LIN {X -0.127,Y -423.917,Z 1358.586,A 0.000,B 0.000,C 90.000,E1 105.536} C_DIS
LIN {X 0.148,Y -443.072,Z 1358.574,A 0.000,B 0.000,C 90.000,E1 103.355} C_DIS
LIN {X 0.036,Y -463.165,Z 1358.563,A 0.000,B 0.000,C 90.000,E1 101.366} C_DIS
LIN {X 0.203,Y -481.163,Z 1358.554,A 0.000,B 0.000,C 90.000,E1 99.726} C_DIS
LIN {X 0.205,Y -483.225,Z 1358.553,A 0.000,B 0.000,C 90.000,E1 99.500} C_DIS
LIN {X -0.191,Y -484.795,Z 1358.552,A 0.000,B 0.000,C 90.000,E1 99.321} C_DIS
LIN {X 0.175,Y -486.110,Z 1358.550,A 0.000,B 0.000,C 90.000,E1 99.029} C_DIS
LIN {X -0.014,Y -487.078,Z 1358.549,A 0.000,B 0.000,C 90.000,E1 98.803} C_DIS
LIN {X 0.255,Y -488.153,Z 1358.546,A 0.000,B 0.000,C 90.000,E1 98.276} C_DIS
LIN {X -0.026,Y -488.220,Z 1358.543,A 0.000,B 0.000,C 90.000,E1 97.814} C_DIS
LIN {X 0.184,Y -487.293,Z 1358.541,A 0.000,B 0.000,C 90.000,E1 97.296} C_DIS
LIN {X -0.088,Y -485.213,Z 1358.538,A 0.000,B 0.000,C 90.000,E1 96.834} C_DIS
LIN {X 0.116,Y -481.753,Z 1358.535,A 0.000,B 0.000,C 90.000,E1 96.315} C_DIS
LIN {X 0.079,Y -471.298,Z 1358.527,A 0.000,B 0.000,C 90.000,E1 94.821} C_DIS
LIN {X -0.125,Y -461.369,Z 1358.518,A 0.000,B 0.000,C 90.000,E1 93.326} C_DIS
LIN {X -0.174,Y -441.725,Z 1358.501,A 0.000,B 0.000,C 90.000,E1 90.229} C_DIS
LIN {X 0.004,Y -428.339,Z 1358.488,A 0.000,B 0.000,C 90.000,E1 87.822} C_DIS
LIN {X 0.068,Y -418.056,Z 1358.477,A 0.000,B 0.000,C 90.000,E1 85.927} C_DIS
LIN {X -0.091,Y -407.688,Z 1358.467,A 0.000,B 0.000,C 90.000,E1 84.033} C_DIS
LIN {X -0.013,Y -398.629,Z 1358.458,A 0.000,B 0.000,C 90.000,E1 82.356} C_DIS
LIN {X -0.094,Y -389.359,Z 1358.448,A 0.000,B 0.000,C 90.000,E1 80.679} C_DIS
LIN {X 0.168,Y -379.910,Z 1358.439,A 0.000,B 0.000,C 90.000,E1 78.926} C_DIS
LIN {X -0.108,Y -370.271,Z 1358.429,A 0.000,B 0.000,C 90.000,E1 77.229} C_DIS
LIN {X -0.144,Y -358.777,Z 1358.417,A 0.000,B 0.000,C 90.000,E1 75.172} C_DIS
LIN {X 0.162,Y -348.864,Z 1358.407,A 0.000,B 0.000,C 90.000,E1 73.323} C_DIS
LIN {X -0.054,Y -337.184,Z 1358.396,A 0.000,B 0.000,C 90.000,E1 71.221} C_DIS
LIN {X -0.015,Y -323.949,Z 1358.382,A 0.000,B 0.000,C 90.000,E1 68.720} C_DIS
LIN {X -0.098,Y -308.256,Z 1358.364,A 0.000,B 0.000,C 90.000,E1 65.537} C_DIS
LIN {X -0.142,Y -298.262,Z 1358.351,A 0.000,B 0.000,C 90.000,E1 63.256} C_DIS
LIN {X 0.106,Y -288.081,Z 1358.336,A 0.000,B 0.000,C 90.000,E1 60.539} C_DIS
LIN {X -0.039,Y -281.281,Z 1358.325,A 0.000,B 0.000,C 90.000,E1 58.535} C_DIS
LIN {X -0.059,Y -271.116,Z 1358.306,A 0.000,B 0.000,C 90.000,E1 55.102} C_DIS
LIN {X 0.096,Y -263.450,Z 1358.291,A 0.000,B 0.000,C 90.000,E1 52.271} C_DIS
LIN {X 0.038,Y -254.301,Z 1358.271,A 0.000,B 0.000,C 90.000,E1 48.728} C_DIS
LIN {X 0.156,Y -247.369,Z 1358.255,A 0.000,B 0.000,C 90.000,E1 45.810} C_DIS
LIN {X 0.070,Y -239.383,Z 1358.234,A 0.000,B 0.000,C 90.000,E1 42.162} C_DIS
LIN {X -0.044,Y -232.253,Z 1358.214,A 0.000,B 0.000,C 90.000,E1 38.463} C_DIS
LIN {X -0.076,Y -225.922,Z 1358.193,A 0.000,B 0.000,C 90.000,E1 34.692} C_DIS
LIN {X -0.007,Y -220.570,Z 1358.171,A 0.000,B 0.000,C 90.000,E1 30.846} C_DIS
LIN {X -0.100,Y -216.212,Z 1358.150,A 0.000,B 0.000,C 90.000,E1 27.001} C_DIS
LIN {X 0.020,Y -212.299,Z 1358.124,A 0.000,B 0.000,C 90.000,E1 22.280} C_DIS
LIN {X -0.044,Y -209.772,Z 1358.102,A 0.000,B 0.000,C 90.000,E1 18.362} C_DIS
LIN {X -0.011,Y -207.919,Z 1358.084,A 0.000,B 0.000,C 90.000,E1 15.190} C_DIS
LIN {X 0.102,Y -205.787,Z 1358.062,A 0.000,B 0.000,C 90.000,E1 11.186} C_DIS
LIN {X -0.089,Y -204.193,Z 1358.045,A 0.000,B 0.000,C 90.000,E1 8.049} C_DIS
LIN {X 0.006,Y -202.797,Z 1358.027,A 0.000,B 0.000,C 90.000,E1 4.821} C_DIS
LIN {X -0.036,Y -200.987,Z 1357.997,A 0.000,B 0.000,C 90.000,E1 359.542} C_DIS
LIN {X -0.090,Y -200.235,Z 1357.966,A 0.000,B 0.000,C 90.000,E1 353.913} C_DIS
LIN {X -0.015,Y -201.594,Z 1357.921,A 0.000,B 0.000,C 90.000,E1 345.825} C_DIS
LIN {X 0.033,Y -204.564,Z 1357.890,A 0.000,B 0.000,C 90.000,E1 340.188} C_DIS
LIN {X 0.003,Y -208.549,Z 1357.863,A 0.000,B 0.000,C 90.000,E1 335.409} C_DIS
LIN {X 0.071,Y -213.049,Z 1357.841,A 0.000,B 0.000,C 90.000,E1 331.435} C_DIS
LIN {X 0.022,Y -218.800,Z 1357.820,A 0.000,B 0.000,C 90.000,E1 327.533} C_DIS
LIN {X -0.119,Y -225.621,Z 1357.798,A 0.000,B 0.000,C 90.000,E1 323.703} C_DIS
LIN {X -0.088,Y -232.011,Z 1357.781,A 0.000,B 0.000,C 90.000,E1 320.642} C_DIS
LIN {X -0.106,Y -239.229,Z 1357.765,A 0.000,B 0.000,C 90.000,E1 317.634} C_DIS
LIN {X 0.024,Y -248.202,Z 1357.746,A 0.000,B 0.000,C 90.000,E1 314.271} C_DIS
LIN {X -0.125,Y -256.103,Z 1357.732,A 0.000,B 0.000,C 90.000,E1 311.757} C_DIS
LIN {X -0.027,Y -266.363,Z 1357.716,A 0.000,B 0.000,C 90.000,E1 308.874} C_DIS
LIN {X -0.018,Y -279.522,Z 1357.698,A 0.000,B 0.000,C 90.000,E1 305.724} C_DIS
LIN {X 0.063,Y -287.690,Z 1357.689,A 0.000,B 0.000,C 90.000,E1 303.992} C_DIS
LIN {X -0.121,Y -296.776,Z 1357.680,A 0.000,B 0.000,C 90.000,E1 302.339} C_DIS
LIN {X -0.078,Y -306.973,Z 1357.670,A 0.000,B 0.000,C 90.000,E1 300.669} C_DIS
LIN {X 0.082,Y -316.117,Z 1357.663,A 0.000,B 0.000,C 90.000,E1 299.333} C_DIS
LIN {X 0.050,Y -336.742,Z 1357.649,A 0.000,B 0.000,C 90.000,E1 296.796} C_DIS
LIN {X -0.056,Y -352.620,Z 1357.639,A 0.000,B 0.000,C 90.000,E1 295.027} C_DIS
LIN {X 0.023,Y -365.723,Z 1357.631,A 0.000,B 0.000,C 90.000,E1 293.567} C_DIS
LIN {X 0.066,Y -375.959,Z 1357.625,A 0.000,B 0.000,C 90.000,E1 292.408} C_DIS
LIN {X -0.001,Y -388.536,Z 1357.616,A 0.000,B 0.000,C 90.000,E1 290.972} C_DIS
LIN {X -0.014,Y -403.296,Z 1357.607,A 0.000,B 0.000,C 90.000,E1 289.268} C_DIS
LIN {X 0.119,Y -417.975,Z 1357.598,A 0.000,B 0.000,C 90.000,E1 287.583} C_DIS
LIN {X 0.090,Y -427.465,Z 1357.592,A 0.000,B 0.000,C 90.000,E1 286.496} C_DIS
LIN {X -0.127,Y -434.044,Z 1357.587,A 0.000,B 0.000,C 90.000,E1 285.717} C_DIS
LIN {X 0.011,Y -440.022,Z 1357.583,A 0.000,B 0.000,C 90.000,E1 284.898} C_DIS
LIN {X -0.102,Y -445.273,Z 1357.578,A 0.000,B 0.000,C 90.000,E1 284.120} C_DIS
LIN {X 0.150,Y -449.712,Z 1357.574,A 0.000,B 0.000,C 90.000,E1 283.300} C_DIS
LIN {X 0.014,Y -453.341,Z 1357.570,A 0.000,B 0.000,C 90.000,E1 282.535} C_DIS
LIN {X -0.097,Y -456.212,Z 1357.565,A 0.000,B 0.000,C 90.000,E1 281.771} C_DIS
LIN {X -0.012,Y -457.679,Z 1357.563,A 0.000,B 0.000,C 90.000,E1 281.243} C_DIS
LIN {X 0.082,Y -458.764,Z 1357.560,A 0.000,B 0.000,C 90.000,E1 280.715} C_DIS
LIN {X 0.100,Y -459.438,Z 1357.557,A 0.000,B 0.000,C 90.000,E1 280.197} C_DIS
LIN {X 0.207,Y -459.649,Z 1357.554,A 0.000,B 0.000,C 90.000,E1 279.670} C_DIS
LIN {X -0.212,Y -459.367,Z 1357.551,A 0.000,B 0.000,C 90.000,E1 279.208} C_DIS
LIN {X -0.104,Y -458.592,Z 1357.548,A 0.000,B 0.000,C 90.000,E1 278.681} C_DIS
LIN {X -0.068,Y -457.352,Z 1357.545,A 0.000,B 0.000,C 90.000,E1 278.163} C_DIS
LIN {X -0.035,Y -455.526,Z 1357.542,A 0.000,B 0.000,C 90.000,E1 277.644} C_DIS
LIN {X -0.006,Y -453.175,Z 1357.540,A 0.000,B 0.000,C 90.000,E1 277.125} C_DIS
LIN {X 0.005,Y -450.289,Z 1357.537,A 0.000,B 0.000,C 90.000,E1 276.606} C_DIS
LIN {X 0.002,Y -446.827,Z 1357.534,A 0.000,B 0.000,C 90.000,E1 276.087} C_DIS
LIN {X -0.019,Y -442.576,Z 1357.531,A 0.000,B 0.000,C 90.000,E1 275.568} C_DIS
LIN {X -0.063,Y -437.339,Z 1357.528,A 0.000,B 0.000,C 90.000,E1 275.049} C_DIS
LIN {X 0.120,Y -431.246,Z 1357.525,A 0.000,B 0.000,C 90.000,E1 274.531} C_DIS
LIN {X -0.098,Y -424.898,Z 1357.523,A 0.000,B 0.000,C 90.000,E1 274.131} C_DIS
LIN {X 0.152,Y -418.457,Z 1357.521,A 0.000,B 0.000,C 90.000,E1 273.726} C_DIS
LIN {X -0.130,Y -412.038,Z 1357.519,A 0.000,B 0.000,C 90.000,E1 273.440} C_DIS
LIN {X 0.208,Y -405.345,Z 1357.517,A 0.000,B 0.000,C 90.000,E1 273.094} C_DIS
LIN {X -0.065,Y -395.236,Z 1357.515,A 0.000,B 0.000,C 90.000,E1 272.751} C_DIS
LIN {X 0.029,Y -388.350,Z 1357.514,A 0.000,B 0.000,C 90.000,E1 272.522} C_DIS
LIN {X -0.051,Y -381.280,Z 1357.513,A 0.000,B 0.000,C 90.000,E1 272.350} C_DIS
LIN {X 0.050,Y -373.704,Z 1357.512,A 0.000,B 0.000,C 90.000,E1 272.178} C_DIS
LIN {X -0.014,Y -364.873,Z 1357.511,A 0.000,B 0.000,C 90.000,E1 272.064} C_DIS
LIN {X -0.163,Y -352.105,Z 1357.511,A 0.000,B 0.000,C 90.000,E1 271.949} C_DIS
LIN {X 0.082,Y -339.041,Z 1357.510,A 0.000,B 0.000,C 90.000,E1 271.835} C_DIS
LIN {X 0.019,Y -330.015,Z 1357.510,A 0.000,B 0.000,C 90.000,E1 271.835} C_DIS
LIN {X -0.009,Y -181.290,Z 1357.510,A 0.000,B 0.000,C 90.000,E1 271.835} C_DIS
LIN {X 0.038,Y -181.580,Z 1357.502,A 0.000,B 0.000,C 90.000,E1 270.286} C_DIS
LIN {X -0.002,Y -180.908,Z 1357.475,A 0.000,B 0.000,C 90.000,E1 265.584} C_DIS
LIN {X 0.055,Y -180.783,Z 1357.471,A 0.000,B 0.000,C 90.000,E1 264.723} C_DIS
LIN {X -0.050,Y -178.880,Z 1357.443,A 0.000,B 0.000,C 90.000,E1 259.690} C_DIS
LIN {X 0.026,Y -175.923,Z 1357.414,A 0.000,B 0.000,C 90.000,E1 254.574} C_DIS
LIN {X -0.084,Y -174.622,Z 1357.405,A 0.000,B 0.000,C 90.000,E1 252.906} C_DIS
LIN {X 0.008,Y -171.603,Z 1357.381,A 0.000,B 0.000,C 90.000,E1 248.592} C_DIS
LIN {X -0.004,Y -167.825,Z 1357.357,A 0.000,B 0.000,C 90.000,E1 244.280} C_DIS
LIN {X 0.014,Y -166.549,Z 1357.347,A 0.000,B 0.000,C 90.000,E1 242.538} C_DIS
LIN {X -0.076,Y -162.546,Z 1357.323,A 0.000,B 0.000,C 90.000,E1 238.201} C_DIS
LIN {X -0.016,Y -161.223,Z 1357.313,A 0.000,B 0.000,C 90.000,E1 236.421} C_DIS
LIN {X 0.020,Y -157.229,Z 1357.289,A 0.000,B 0.000,C 90.000,E1 231.984} C_DIS
LIN {X 0.043,Y -155.955,Z 1357.279,A 0.000,B 0.000,C 90.000,E1 230.194} C_DIS
LIN {X 0.001,Y -152.207,Z 1357.254,A 0.000,B 0.000,C 90.000,E1 225.729} C_DIS
LIN {X 0.022,Y -150.452,Z 1357.239,A 0.000,B 0.000,C 90.000,E1 223.014} C_DIS
LIN {X 0.048,Y -147.178,Z 1357.214,A 0.000,B 0.000,C 90.000,E1 218.463} C_DIS
LIN {X 0.015,Y -145.196,Z 1357.193,A 0.000,B 0.000,C 90.000,E1 214.818} C_DIS
LIN {X 0.050,Y -142.335,Z 1357.163,A 0.000,B 0.000,C 90.000,E1 209.283} C_DIS
LIN {X -0.021,Y -141.723,Z 1357.152,A 0.000,B 0.000,C 90.000,E1 207.462} C_DIS
LIN {X -0.039,Y -139.479,Z 1357.116,A 0.000,B 0.000,C 90.000,E1 200.972} C_DIS
LIN {X -0.049,Y -138.976,Z 1357.101,A 0.000,B 0.000,C 90.000,E1 198.181} C_DIS
LIN {X 0.072,Y -138.331,Z 1357.054,A 0.000,B 0.000,C 90.000,E1 189.726} C_DIS
LIN {X -0.064,Y -139.432,Z 1357.007,A 0.000,B 0.000,C 90.000,E1 181.375} C_DIS
LIN {X 0.015,Y -140.958,Z 1356.976,A 0.000,B 0.000,C 90.000,E1 175.755} C_DIS
LIN {X -0.034,Y -142.713,Z 1356.956,A 0.000,B 0.000,C 90.000,E1 172.064} C_DIS
LIN {X 0.065,Y -145.090,Z 1356.930,A 0.000,B 0.000,C 90.000,E1 167.409} C_DIS
LIN {X 0.061,Y -147.715,Z 1356.910,A 0.000,B 0.000,C 90.000,E1 163.740} C_DIS
LIN {X 0.002,Y -150.372,Z 1356.890,A 0.000,B 0.000,C 90.000,E1 160.115} C_DIS
LIN {X 0.020,Y -153.800,Z 1356.869,A 0.000,B 0.000,C 90.000,E1 156.485} C_DIS
LIN {X 0.080,Y -157.211,Z 1356.849,A 0.000,B 0.000,C 90.000,E1 152.871} C_DIS
LIN {X 0.021,Y -161.376,Z 1356.830,A 0.000,B 0.000,C 90.000,E1 149.331} C_DIS
LIN {X 0.032,Y -165.578,Z 1356.810,A 0.000,B 0.000,C 90.000,E1 145.801} C_DIS
LIN {X 0.018,Y -170.499,Z 1356.791,A 0.000,B 0.000,C 90.000,E1 142.316} C_DIS
LIN {X 0.064,Y -175.379,Z 1356.771,A 0.000,B 0.000,C 90.000,E1 138.852} C_DIS
LIN {X -0.074,Y -181.003,Z 1356.753,A 0.000,B 0.000,C 90.000,E1 135.486} C_DIS
LIN {X 0.051,Y -186.431,Z 1356.734,A 0.000,B 0.000,C 90.000,E1 132.081} C_DIS
LIN {X 0.119,Y -191.058,Z 1356.720,A 0.000,B 0.000,C 90.000,E1 129.564} C_DIS
LIN {X 0.042,Y -196.843,Z 1356.702,A 0.000,B 0.000,C 90.000,E1 126.297} C_DIS
LIN {X 0.051,Y -199.194,Z 1356.695,A 0.000,B 0.000,C 90.000,E1 125.105} C_DIS
LIN {X 0.046,Y -308.858,Z 1356.695,A 0.000,B 0.000,C 90.000,E1 125.105} C_DIS
LIN {X -0.191,Y -311.436,Z 1356.695,A 0.000,B 0.000,C 90.000,E1 125.105} C_DIS
LIN {X -0.128,Y -315.472,Z 1356.694,A 0.000,B 0.000,C 90.000,E1 124.898} C_DIS
LIN {X -0.063,Y -317.840,Z 1356.693,A 0.000,B 0.000,C 90.000,E1 124.692} C_DIS
LIN {X 0.014,Y -321.665,Z 1356.690,A 0.000,B 0.000,C 90.000,E1 124.199} C_DIS
LIN {X 0.089,Y -323.434,Z 1356.688,A 0.000,B 0.000,C 90.000,E1 123.865} C_DIS
LIN {X -0.106,Y -324.810,Z 1356.686,A 0.000,B 0.000,C 90.000,E1 123.579} C_DIS
LIN {X -0.011,Y -336.372,Z 1356.669,A 0.000,B 0.000,C 90.000,E1 120.413} C_DIS
LIN {X -0.054,Y -348.165,Z 1356.654,A 0.000,B 0.000,C 90.000,E1 117.641} C_DIS
LIN {X 0.058,Y -361.406,Z 1356.638,A 0.000,B 0.000,C 90.000,E1 114.899} C_DIS
LIN {X 0.156,Y -374.481,Z 1356.625,A 0.000,B 0.000,C 90.000,E1 112.514} C_DIS
LIN {X -0.202,Y -388.879,Z 1356.612,A 0.000,B 0.000,C 90.000,E1 110.248} C_DIS
LIN {X 0.033,Y -404.701,Z 1356.600,A 0.000,B 0.000,C 90.000,E1 107.946} C_DIS
LIN {X 0.154,Y -422.057,Z 1356.587,A 0.000,B 0.000,C 90.000,E1 105.717} C_DIS
LIN {X -0.058,Y -441.070,Z 1356.575,A 0.000,B 0.000,C 90.000,E1 103.592} C_DIS
LIN {X 0.228,Y -461.105,Z 1356.564,A 0.000,B 0.000,C 90.000,E1 101.535} C_DIS
LIN {X -0.165,Y -481.566,Z 1356.554,A 0.000,B 0.000,C 90.000,E1 99.726} C_DIS
LIN {X -0.201,Y -483.525,Z 1356.553,A 0.000,B 0.000,C 90.000,E1 99.500} C_DIS
LIN {X -0.156,Y -485.019,Z 1356.551,A 0.000,B 0.000,C 90.000,E1 99.265} C_DIS
LIN {X 0.212,Y -486.241,Z 1356.550,A 0.000,B 0.000,C 90.000,E1 98.973} C_DIS
LIN {X 0.025,Y -487.133,Z 1356.549,A 0.000,B 0.000,C 90.000,E1 98.746} C_DIS
LIN {X -0.187,Y -488.080,Z 1356.546,A 0.000,B 0.000,C 90.000,E1 98.276} C_DIS
LIN {X 0.015,Y -488.028,Z 1356.543,A 0.000,B 0.000,C 90.000,E1 97.757} C_DIS
LIN {X 0.225,Y -486.975,Z 1356.540,A 0.000,B 0.000,C 90.000,E1 97.239} C_DIS
LIN {X 0.119,Y -486.024,Z 1356.539,A 0.000,B 0.000,C 90.000,E1 97.004} C_DIS
LIN {X -0.047,Y -484.730,Z 1356.538,A 0.000,B 0.000,C 90.000,E1 96.777} C_DIS
LIN {X 0.143,Y -470.717,Z 1356.526,A 0.000,B 0.000,C 90.000,E1 94.759} C_DIS
LIN {X -0.109,Y -460.779,Z 1356.518,A 0.000,B 0.000,C 90.000,E1 93.269} C_DIS
LIN {X 0.073,Y -442.697,Z 1356.502,A 0.000,B 0.000,C 90.000,E1 90.401} C_DIS
LIN {X -0.155,Y -429.271,Z 1356.489,A 0.000,B 0.000,C 90.000,E1 88.051} C_DIS
LIN {X -0.098,Y -419.002,Z 1356.479,A 0.000,B 0.000,C 90.000,E1 86.159} C_DIS
LIN {X -0.196,Y -408.662,Z 1356.468,A 0.000,B 0.000,C 90.000,E1 84.261} C_DIS
LIN {X -0.146,Y -399.649,Z 1356.459,A 0.000,B 0.000,C 90.000,E1 82.591} C_DIS
LIN {X -0.149,Y -390.407,Z 1356.449,A 0.000,B 0.000,C 90.000,E1 80.905} C_DIS
LIN {X 0.070,Y -380.987,Z 1356.440,A 0.000,B 0.000,C 90.000,E1 79.162} C_DIS
LIN {X 0.176,Y -371.371,Z 1356.430,A 0.000,B 0.000,C 90.000,E1 77.409} C_DIS
LIN {X -0.202,Y -359.872,Z 1356.419,A 0.000,B 0.000,C 90.000,E1 75.408} C_DIS
LIN {X 0.127,Y -349.982,Z 1356.409,A 0.000,B 0.000,C 90.000,E1 73.559} C_DIS
LIN {X -0.057,Y -338.318,Z 1356.397,A 0.000,B 0.000,C 90.000,E1 71.456} C_DIS
LIN {X 0.046,Y -326.707,Z 1356.385,A 0.000,B 0.000,C 90.000,E1 69.263} C_DIS
LIN {X -0.153,Y -309.304,Z 1356.365,A 0.000,B 0.000,C 90.000,E1 65.793} C_DIS
LIN {X 0.089,Y -299.177,Z 1356.353,A 0.000,B 0.000,C 90.000,E1 63.461} C_DIS
LIN {X 0.095,Y -288.907,Z 1356.338,A 0.000,B 0.000,C 90.000,E1 60.795} C_DIS
LIN {X -0.001,Y -283.110,Z 1356.328,A 0.000,B 0.000,C 90.000,E1 59.125} C_DIS
LIN {X 0.107,Y -272.805,Z 1356.309,A 0.000,B 0.000,C 90.000,E1 55.674} C_DIS
LIN {X 0.065,Y -263.208,Z 1356.290,A 0.000,B 0.000,C 90.000,E1 52.190} C_DIS
LIN {X 0.002,Y -254.112,Z 1356.270,A 0.000,B 0.000,C 90.000,E1 48.647} C_DIS
LIN {X 0.117,Y -247.203,Z 1356.254,A 0.000,B 0.000,C 90.000,E1 45.729} C_DIS
LIN {X 0.026,Y -239.269,Z 1356.234,A 0.000,B 0.000,C 90.000,E1 42.081} C_DIS
LIN {X -0.090,Y -232.167,Z 1356.213,A 0.000,B 0.000,C 90.000,E1 38.382} C_DIS
LIN {X -0.127,Y -225.863,Z 1356.192,A 0.000,B 0.000,C 90.000,E1 34.612} C_DIS
LIN {X 0.014,Y -220.556,Z 1356.171,A 0.000,B 0.000,C 90.000,E1 30.747} C_DIS
LIN {X -0.005,Y -215.494,Z 1356.145,A 0.000,B 0.000,C 90.000,E1 26.104} C_DIS
LIN {X 0.000,Y -211.802,Z 1356.119,A 0.000,B 0.000,C 90.000,E1 21.408} C_DIS
LIN {X 0.082,Y -209.816,Z 1356.101,A 0.000,B 0.000,C 90.000,E1 18.236} C_DIS
LIN {X 0.057,Y -207.959,Z 1356.084,A 0.000,B 0.000,C 90.000,E1 15.079} C_DIS
LIN {X -0.025,Y -205.804,Z 1356.062,A 0.000,B 0.000,C 90.000,E1 11.130} C_DIS
LIN {X 0.029,Y -203.803,Z 1356.040,A 0.000,B 0.000,C 90.000,E1 7.125} C_DIS
LIN {X -0.089,Y -202.106,Z 1356.017,A 0.000,B 0.000,C 90.000,E1 3.151} C_DIS
LIN {X -0.056,Y -200.678,Z 1355.988,A 0.000,B 0.000,C 90.000,E1 357.936} C_DIS
LIN {X -0.079,Y -200.375,Z 1355.953,A 0.000,B 0.000,C 90.000,E1 351.489} C_DIS
LIN {X 0.002,Y -202.383,Z 1355.912,A 0.000,B 0.000,C 90.000,E1 344.212} C_DIS
LIN {X 0.030,Y -205.836,Z 1355.881,A 0.000,B 0.000,C 90.000,E1 338.592} C_DIS
LIN {X 0.032,Y -210.370,Z 1355.855,A 0.000,B 0.000,C 90.000,E1 333.819} C_DIS
LIN {X 0.065,Y -215.370,Z 1355.833,A 0.000,B 0.000,C 90.000,E1 329.871} C_DIS
LIN {X -0.056,Y -221.576,Z 1355.811,A 0.000,B 0.000,C 90.000,E1 326.008} C_DIS
LIN {X -0.038,Y -227.334,Z 1355.794,A 0.000,B 0.000,C 90.000,E1 322.924} C_DIS
LIN {X -0.145,Y -233.901,Z 1355.777,A 0.000,B 0.000,C 90.000,E1 319.908} C_DIS
LIN {X 0.041,Y -241.291,Z 1355.760,A 0.000,B 0.000,C 90.000,E1 316.863} C_DIS
LIN {X 0.064,Y -250.485,Z 1355.742,A 0.000,B 0.000,C 90.000,E1 313.542} C_DIS
LIN {X -0.014,Y -258.668,Z 1355.728,A 0.000,B 0.000,C 90.000,E1 311.024} C_DIS
LIN {X -0.072,Y -267.877,Z 1355.714,A 0.000,B 0.000,C 90.000,E1 308.543} C_DIS
LIN {X 0.047,Y -279.652,Z 1355.698,A 0.000,B 0.000,C 90.000,E1 305.724} C_DIS
LIN {X -0.137,Y -289.565,Z 1355.687,A 0.000,B 0.000,C 90.000,E1 303.706} C_DIS
LIN {X -0.054,Y -298.877,Z 1355.678,A 0.000,B 0.000,C 90.000,E1 302.005} C_DIS
LIN {X 0.001,Y -307.086,Z 1355.670,A 0.000,B 0.000,C 90.000,E1 300.669} C_DIS
LIN {X 0.163,Y -316.214,Z 1355.663,A 0.000,B 0.000,C 90.000,E1 299.333} C_DIS
LIN {X -0.005,Y -334.150,Z 1355.651,A 0.000,B 0.000,C 90.000,E1 297.129} C_DIS
LIN {X -0.067,Y -352.771,Z 1355.639,A 0.000,B 0.000,C 90.000,E1 295.027} C_DIS
LIN {X -0.045,Y -365.954,Z 1355.631,A 0.000,B 0.000,C 90.000,E1 293.567} C_DIS
LIN {X 0.071,Y -376.247,Z 1355.624,A 0.000,B 0.000,C 90.000,E1 292.386} C_DIS
LIN {X -0.158,Y -388.803,Z 1355.616,A 0.000,B 0.000,C 90.000,E1 290.972} C_DIS
LIN {X 0.023,Y -401.110,Z 1355.609,A 0.000,B 0.000,C 90.000,E1 289.523} C_DIS
LIN {X -0.145,Y -415.800,Z 1355.599,A 0.000,B 0.000,C 90.000,E1 287.873} C_DIS
LIN {X 0.197,Y -425.376,Z 1355.593,A 0.000,B 0.000,C 90.000,E1 286.732} C_DIS
LIN {X -0.044,Y -432.138,Z 1355.589,A 0.000,B 0.000,C 90.000,E1 285.953} C_DIS
LIN {X 0.081,Y -438.272,Z 1355.584,A 0.000,B 0.000,C 90.000,E1 285.134} C_DIS
LIN {X 0.170,Y -442.080,Z 1355.581,A 0.000,B 0.000,C 90.000,E1 284.592} C_DIS
LIN {X -0.041,Y -447.075,Z 1355.577,A 0.000,B 0.000,C 90.000,E1 283.828} C_DIS
LIN {X -0.203,Y -451.218,Z 1355.572,A 0.000,B 0.000,C 90.000,E1 283.063} C_DIS
LIN {X 0.111,Y -454.614,Z 1355.568,A 0.000,B 0.000,C 90.000,E1 282.243} C_DIS
LIN {X 0.193,Y -456.453,Z 1355.565,A 0.000,B 0.000,C 90.000,E1 281.715} C_DIS
LIN {X -0.169,Y -457.920,Z 1355.562,A 0.000,B 0.000,C 90.000,E1 281.243} C_DIS
LIN {X -0.075,Y -458.991,Z 1355.559,A 0.000,B 0.000,C 90.000,E1 280.715} C_DIS
LIN {X -0.055,Y -459.696,Z 1355.557,A 0.000,B 0.000,C 90.000,E1 280.197} C_DIS
LIN {X 0.055,Y -459.925,Z 1355.554,A 0.000,B 0.000,C 90.000,E1 279.670} C_DIS
LIN {X 0.090,Y -459.619,Z 1355.551,A 0.000,B 0.000,C 90.000,E1 279.151} C_DIS
LIN {X 0.199,Y -458.873,Z 1355.548,A 0.000,B 0.000,C 90.000,E1 278.624} C_DIS
LIN {X -0.217,Y -457.601,Z 1355.545,A 0.000,B 0.000,C 90.000,E1 278.163} C_DIS
LIN {X -0.181,Y -455.830,Z 1355.542,A 0.000,B 0.000,C 90.000,E1 277.644} C_DIS
LIN {X -0.151,Y -453.485,Z 1355.539,A 0.000,B 0.000,C 90.000,E1 277.125} C_DIS
LIN {X -0.136,Y -450.620,Z 1355.537,A 0.000,B 0.000,C 90.000,E1 276.606} C_DIS
LIN {X -0.137,Y -447.151,Z 1355.534,A 0.000,B 0.000,C 90.000,E1 276.087} C_DIS
LIN {X -0.154,Y -442.942,Z 1355.531,A 0.000,B 0.000,C 90.000,E1 275.568} C_DIS
LIN {X -0.195,Y -437.696,Z 1355.528,A 0.000,B 0.000,C 90.000,E1 275.049} C_DIS
LIN {X -0.024,Y -431.649,Z 1355.525,A 0.000,B 0.000,C 90.000,E1 274.531} C_DIS
LIN {X 0.184,Y -425.386,Z 1355.523,A 0.000,B 0.000,C 90.000,E1 274.073} C_DIS
LIN {X -0.022,Y -418.927,Z 1355.521,A 0.000,B 0.000,C 90.000,E1 273.726} C_DIS
LIN {X 0.086,Y -412.492,Z 1355.519,A 0.000,B 0.000,C 90.000,E1 273.383} C_DIS
LIN {X 0.001,Y -405.787,Z 1355.517,A 0.000,B 0.000,C 90.000,E1 273.094} C_DIS
LIN {X 0.130,Y -395.660,Z 1355.515,A 0.000,B 0.000,C 90.000,E1 272.694} C_DIS
LIN {X -0.183,Y -388.690,Z 1355.514,A 0.000,B 0.000,C 90.000,E1 272.522} C_DIS
LIN {X 0.102,Y -381.476,Z 1355.513,A 0.000,B 0.000,C 90.000,E1 272.293} C_DIS
LIN {X -0.176,Y -373.907,Z 1355.512,A 0.000,B 0.000,C 90.000,E1 272.178} C_DIS
LIN {X 0.135,Y -365.143,Z 1355.511,A 0.000,B 0.000,C 90.000,E1 272.007} C_DIS
LIN {X -0.024,Y -351.696,Z 1355.510,A 0.000,B 0.000,C 90.000,E1 271.892} C_DIS
LIN {X -0.055,Y -339.050,Z 1355.510,A 0.000,B 0.000,C 90.000,E1 271.835} C_DIS
LIN {X -0.062,Y -181.293,Z 1355.510,A 0.000,B 0.000,C 90.000,E1 271.835} C_DIS
LIN {X 0.012,Y -181.581,Z 1355.502,A 0.000,B 0.000,C 90.000,E1 270.286} C_DIS
LIN {X -0.028,Y -180.908,Z 1355.475,A 0.000,B 0.000,C 90.000,E1 265.584} C_DIS
LIN {X 0.030,Y -180.780,Z 1355.471,A 0.000,B 0.000,C 90.000,E1 264.723} C_DIS
LIN {X -0.076,Y -178.877,Z 1355.443,A 0.000,B 0.000,C 90.000,E1 259.690} C_DIS
LIN {X 0.000,Y -175.919,Z 1355.414,A 0.000,B 0.000,C 90.000,E1 254.574} C_DIS
LIN {X 0.056,Y -174.615,Z 1355.405,A 0.000,B 0.000,C 90.000,E1 252.851} C_DIS
LIN {X -0.017,Y -171.596,Z 1355.381,A 0.000,B 0.000,C 90.000,E1 248.592} C_DIS
LIN {X -0.028,Y -167.818,Z 1355.357,A 0.000,B 0.000,C 90.000,E1 244.280} C_DIS
LIN {X -0.011,Y -166.542,Z 1355.347,A 0.000,B 0.000,C 90.000,E1 242.538} C_DIS
LIN {X -0.100,Y -162.538,Z 1355.323,A 0.000,B 0.000,C 90.000,E1 238.201} C_DIS
LIN {X -0.040,Y -161.214,Z 1355.313,A 0.000,B 0.000,C 90.000,E1 236.421} C_DIS
LIN {X -0.004,Y -157.223,Z 1355.289,A 0.000,B 0.000,C 90.000,E1 231.984} C_DIS
LIN {X 0.019,Y -155.948,Z 1355.279,A 0.000,B 0.000,C 90.000,E1 230.194} C_DIS
LIN {X -0.022,Y -152.201,Z 1355.254,A 0.000,B 0.000,C 90.000,E1 225.729} C_DIS
LIN {X -0.001,Y -150.446,Z 1355.239,A 0.000,B 0.000,C 90.000,E1 223.014} C_DIS
LIN {X 0.026,Y -147.173,Z 1355.214,A 0.000,B 0.000,C 90.000,E1 218.463} C_DIS
LIN {X -0.007,Y -145.190,Z 1355.193,A 0.000,B 0.000,C 90.000,E1 214.818} C_DIS
LIN {X 0.027,Y -142.331,Z 1355.163,A 0.000,B 0.000,C 90.000,E1 209.283} C_DIS
LIN {X -0.043,Y -141.721,Z 1355.152,A 0.000,B 0.000,C 90.000,E1 207.462} C_DIS
LIN {X -0.061,Y -139.477,Z 1355.116,A 0.000,B 0.000,C 90.000,E1 200.972} C_DIS
LIN {X -0.072,Y -138.974,Z 1355.101,A 0.000,B 0.000,C 90.000,E1 198.181} C_DIS
LIN {X 0.050,Y -138.331,Z 1355.054,A 0.000,B 0.000,C 90.000,E1 189.726} C_DIS
LIN {X 0.053,Y -139.433,Z 1355.007,A 0.000,B 0.000,C 90.000,E1 181.318} C_DIS
LIN {X -0.007,Y -140.961,Z 1354.976,A 0.000,B 0.000,C 90.000,E1 175.755} C_DIS
LIN {X -0.057,Y -142.717,Z 1354.956,A 0.000,B 0.000,C 90.000,E1 172.064} C_DIS
LIN {X 0.042,Y -145.096,Z 1354.930,A 0.000,B 0.000,C 90.000,E1 167.409} C_DIS
LIN {X 0.037,Y -147.720,Z 1354.910,A 0.000,B 0.000,C 90.000,E1 163.740} C_DIS
LIN {X -0.021,Y -150.379,Z 1354.890,A 0.000,B 0.000,C 90.000,E1 160.115} C_DIS
LIN {X -0.004,Y -153.809,Z 1354.869,A 0.000,B 0.000,C 90.000,E1 156.485} C_DIS
LIN {X 0.055,Y -157.221,Z 1354.849,A 0.000,B 0.000,C 90.000,E1 152.871} C_DIS
LIN {X -0.004,Y -161.387,Z 1354.830,A 0.000,B 0.000,C 90.000,E1 149.331} C_DIS
LIN {X 0.007,Y -165.589,Z 1354.810,A 0.000,B 0.000,C 90.000,E1 145.801} C_DIS
LIN {X -0.007,Y -170.512,Z 1354.791,A 0.000,B 0.000,C 90.000,E1 142.316} C_DIS
LIN {X 0.038,Y -175.391,Z 1354.771,A 0.000,B 0.000,C 90.000,E1 138.852} C_DIS
LIN {X -0.100,Y -181.016,Z 1354.753,A 0.000,B 0.000,C 90.000,E1 135.486} C_DIS
LIN {X 0.024,Y -186.446,Z 1354.734,A 0.000,B 0.000,C 90.000,E1 132.081} C_DIS
LIN {X 0.092,Y -191.070,Z 1354.720,A 0.000,B 0.000,C 90.000,E1 129.564} C_DIS
LIN {X 0.015,Y -196.858,Z 1354.702,A 0.000,B 0.000,C 90.000,E1 126.297} C_DIS
LIN {X 0.049,Y -199.195,Z 1354.695,A 0.000,B 0.000,C 90.000,E1 125.105} C_DIS
LIN {X 0.037,Y -309.043,Z 1354.695,A 0.000,B 0.000,C 90.000,E1 125.105} C_DIS
LIN {X -0.035,Y -315.193,Z 1354.694,A 0.000,B 0.000,C 90.000,E1 124.898} C_DIS
LIN {X -0.107,Y -317.898,Z 1354.693,A 0.000,B 0.000,C 90.000,E1 124.692} C_DIS
LIN {X -0.003,Y -321.662,Z 1354.690,A 0.000,B 0.000,C 90.000,E1 124.199} C_DIS
LIN {X 0.071,Y -323.427,Z 1354.688,A 0.000,B 0.000,C 90.000,E1 123.865} C_DIS
LIN {X -0.123,Y -324.801,Z 1354.686,A 0.000,B 0.000,C 90.000,E1 123.579} C_DIS
LIN {X -0.030,Y -336.362,Z 1354.669,A 0.000,B 0.000,C 90.000,E1 120.413} C_DIS
LIN {X -0.074,Y -348.157,Z 1354.653,A 0.000,B 0.000,C 90.000,E1 117.641} C_DIS
LIN {X 0.038,Y -361.399,Z 1354.638,A 0.000,B 0.000,C 90.000,E1 114.899} C_DIS
LIN {X 0.135,Y -374.475,Z 1354.625,A 0.000,B 0.000,C 90.000,E1 112.514} C_DIS
LIN {X -0.224,Y -388.875,Z 1354.612,A 0.000,B 0.000,C 90.000,E1 110.248} C_DIS
LIN {X 0.010,Y -404.699,Z 1354.600,A 0.000,B 0.000,C 90.000,E1 107.946} C_DIS
LIN {X 0.131,Y -422.057,Z 1354.587,A 0.000,B 0.000,C 90.000,E1 105.717} C_DIS
LIN {X -0.082,Y -441.072,Z 1354.575,A 0.000,B 0.000,C 90.000,E1 103.592} C_DIS
LIN {X 0.204,Y -461.108,Z 1354.564,A 0.000,B 0.000,C 90.000,E1 101.535} C_DIS
LIN {X -0.190,Y -481.545,Z 1354.554,A 0.000,B 0.000,C 90.000,E1 99.726} C_DIS
LIN {X -0.236,Y -483.486,Z 1354.553,A 0.000,B 0.000,C 90.000,E1 99.500} C_DIS
LIN {X -0.203,Y -484.963,Z 1354.551,A 0.000,B 0.000,C 90.000,E1 99.265} C_DIS
LIN {X 0.164,Y -486.165,Z 1354.550,A 0.000,B 0.000,C 90.000,E1 98.973} C_DIS
LIN {X -0.023,Y -487.038,Z 1354.549,A 0.000,B 0.000,C 90.000,E1 98.746} C_DIS
LIN {X 0.246,Y -487.953,Z 1354.546,A 0.000,B 0.000,C 90.000,E1 98.219} C_DIS
LIN {X -0.034,Y -487.873,Z 1354.543,A 0.000,B 0.000,C 90.000,E1 97.757} C_DIS
LIN {X 0.175,Y -486.788,Z 1354.540,A 0.000,B 0.000,C 90.000,E1 97.239} C_DIS
LIN {X 0.068,Y -485.819,Z 1354.539,A 0.000,B 0.000,C 90.000,E1 97.004} C_DIS
LIN {X -0.098,Y -484.503,Z 1354.538,A 0.000,B 0.000,C 90.000,E1 96.777} C_DIS
LIN {X 0.088,Y -470.445,Z 1354.526,A 0.000,B 0.000,C 90.000,E1 94.759} C_DIS
LIN {X -0.167,Y -460.527,Z 1354.518,A 0.000,B 0.000,C 90.000,E1 93.269} C_DIS
LIN {X -0.180,Y -443.975,Z 1354.504,A 0.000,B 0.000,C 90.000,E1 90.688} C_DIS
LIN {X 0.204,Y -429.015,Z 1354.489,A 0.000,B 0.000,C 90.000,E1 87.993} C_DIS
LIN {X -0.171,Y -418.755,Z 1354.479,A 0.000,B 0.000,C 90.000,E1 86.159} C_DIS
LIN {X 0.134,Y -408.436,Z 1354.468,A 0.000,B 0.000,C 90.000,E1 84.204} C_DIS
LIN {X 0.172,Y -399.411,Z 1354.459,A 0.000,B 0.000,C 90.000,E1 82.534} C_DIS
LIN {X 0.156,Y -390.185,Z 1354.449,A 0.000,B 0.000,C 90.000,E1 80.849} C_DIS
LIN {X -0.013,Y -380.771,Z 1354.440,A 0.000,B 0.000,C 90.000,E1 79.162} C_DIS
LIN {X 0.091,Y -371.148,Z 1354.430,A 0.000,B 0.000,C 90.000,E1 77.409} C_DIS
LIN {X 0.060,Y -359.627,Z 1354.419,A 0.000,B 0.000,C 90.000,E1 75.353} C_DIS
LIN {X 0.039,Y -349.755,Z 1354.409,A 0.000,B 0.000,C 90.000,E1 73.559} C_DIS
LIN {X -0.147,Y -338.092,Z 1354.397,A 0.000,B 0.000,C 90.000,E1 71.456} C_DIS
LIN {X -0.077,Y -324.859,Z 1354.383,A 0.000,B 0.000,C 90.000,E1 68.954} C_DIS
LIN {X 0.074,Y -307.618,Z 1354.363,A 0.000,B 0.000,C 90.000,E1 65.409} C_DIS
LIN {X 0.012,Y -297.646,Z 1354.351,A 0.000,B 0.000,C 90.000,E1 63.127} C_DIS
LIN {X -0.012,Y -287.548,Z 1354.336,A 0.000,B 0.000,C 90.000,E1 60.461} C_DIS
LIN {X 0.079,Y -280.830,Z 1354.325,A 0.000,B 0.000,C 90.000,E1 58.408} C_DIS
LIN {X 0.038,Y -270.743,Z 1354.305,A 0.000,B 0.000,C 90.000,E1 54.975} C_DIS
LIN {X -0.031,Y -263.140,Z 1354.290,A 0.000,B 0.000,C 90.000,E1 52.190} C_DIS
LIN {X 0.075,Y -254.080,Z 1354.270,A 0.000,B 0.000,C 90.000,E1 48.609} C_DIS
LIN {X 0.026,Y -245.532,Z 1354.250,A 0.000,B 0.000,C 90.000,E1 45.000} C_DIS
LIN {X 0.062,Y -237.820,Z 1354.230,A 0.000,B 0.000,C 90.000,E1 41.310} C_DIS
LIN {X -0.066,Y -230.882,Z 1354.209,A 0.000,B 0.000,C 90.000,E1 37.604} C_DIS
LIN {X 0.044,Y -224.783,Z 1354.188,A 0.000,B 0.000,C 90.000,E1 33.785} C_DIS
LIN {X 0.034,Y -219.668,Z 1354.167,A 0.000,B 0.000,C 90.000,E1 29.951} C_DIS
LIN {X 0.075,Y -214.886,Z 1354.141,A 0.000,B 0.000,C 90.000,E1 25.283} C_DIS
LIN {X -0.024,Y -211.380,Z 1354.115,A 0.000,B 0.000,C 90.000,E1 20.610} C_DIS
LIN {X -0.062,Y -208.945,Z 1354.093,A 0.000,B 0.000,C 90.000,E1 16.677} C_DIS
LIN {X 0.039,Y -207.114,Z 1354.075,A 0.000,B 0.000,C 90.000,E1 13.480} C_DIS
LIN {X -0.002,Y -205.407,Z 1354.057,A 0.000,B 0.000,C 90.000,E1 10.310} C_DIS
LIN {X 0.003,Y -203.437,Z 1354.035,A 0.000,B 0.000,C 90.000,E1 6.315} C_DIS
LIN {X 0.044,Y -201.559,Z 1354.008,A 0.000,B 0.000,C 90.000,E1 1.489} C_DIS
LIN {X -0.080,Y -200.457,Z 1353.979,A 0.000,B 0.000,C 90.000,E1 356.331} C_DIS
LIN {X -0.020,Y -200.631,Z 1353.944,A 0.000,B 0.000,C 90.000,E1 349.859} C_DIS
LIN {X 0.032,Y -203.317,Z 1353.903,A 0.000,B 0.000,C 90.000,E1 342.598} C_DIS
LIN {X 0.040,Y -206.611,Z 1353.877,A 0.000,B 0.000,C 90.000,E1 337.794} C_DIS
LIN {X -0.046,Y -210.531,Z 1353.855,A 0.000,B 0.000,C 90.000,E1 333.845} C_DIS
LIN {X 0.086,Y -215.535,Z 1353.833,A 0.000,B 0.000,C 90.000,E1 329.871} C_DIS
LIN {X -0.029,Y -221.746,Z 1353.811,A 0.000,B 0.000,C 90.000,E1 326.008} C_DIS
LIN {X -0.005,Y -227.513,Z 1353.794,A 0.000,B 0.000,C 90.000,E1 322.924} C_DIS
LIN {X -0.107,Y -234.055,Z 1353.777,A 0.000,B 0.000,C 90.000,E1 319.908} C_DIS
LIN {X -0.092,Y -241.414,Z 1353.760,A 0.000,B 0.000,C 90.000,E1 316.905} C_DIS
LIN {X 0.113,Y -250.606,Z 1353.742,A 0.000,B 0.000,C 90.000,E1 313.542} C_DIS
LIN {X 0.038,Y -258.772,Z 1353.728,A 0.000,B 0.000,C 90.000,E1 311.024} C_DIS
LIN {X -0.015,Y -267.972,Z 1353.714,A 0.000,B 0.000,C 90.000,E1 308.543} C_DIS
LIN {X 0.108,Y -279.775,Z 1353.699,A 0.000,B 0.000,C 90.000,E1 305.724} C_DIS
LIN {X -0.070,Y -289.667,Z 1353.687,A 0.000,B 0.000,C 90.000,E1 303.706} C_DIS
LIN {X 0.017,Y -299.000,Z 1353.678,A 0.000,B 0.000,C 90.000,E1 302.005} C_DIS
LIN {X 0.075,Y -307.210,Z 1353.670,A 0.000,B 0.000,C 90.000,E1 300.669} C_DIS
LIN {X -0.190,Y -316.305,Z 1353.663,A 0.000,B 0.000,C 90.000,E1 299.411} C_DIS
LIN {X -0.034,Y -331.535,Z 1353.653,A 0.000,B 0.000,C 90.000,E1 297.462} C_DIS
LIN {X -0.080,Y -350.164,Z 1353.641,A 0.000,B 0.000,C 90.000,E1 295.335} C_DIS
LIN {X -0.190,Y -363.294,Z 1353.633,A 0.000,B 0.000,C 90.000,E1 293.898} C_DIS
LIN {X 0.017,Y -376.294,Z 1353.625,A 0.000,B 0.000,C 90.000,E1 292.408} C_DIS
LIN {X -0.067,Y -388.769,Z 1353.616,A 0.000,B 0.000,C 90.000,E1 290.972} C_DIS
LIN {X 0.116,Y -401.048,Z 1353.609,A 0.000,B 0.000,C 90.000,E1 289.523} C_DIS
LIN {X -0.050,Y -415.758,Z 1353.599,A 0.000,B 0.000,C 90.000,E1 287.873} C_DIS
LIN {X -0.236,Y -425.325,Z 1353.593,A 0.000,B 0.000,C 90.000,E1 286.804} C_DIS
LIN {X -0.065,Y -432.074,Z 1353.589,A 0.000,B 0.000,C 90.000,E1 285.969} C_DIS
LIN {X 0.180,Y -438.275,Z 1353.584,A 0.000,B 0.000,C 90.000,E1 285.134} C_DIS
LIN {X 0.049,Y -443.835,Z 1353.580,A 0.000,B 0.000,C 90.000,E1 284.356} C_DIS
LIN {X -0.142,Y -448.571,Z 1353.575,A 0.000,B 0.000,C 90.000,E1 283.592} C_DIS
LIN {X 0.145,Y -452.509,Z 1353.571,A 0.000,B 0.000,C 90.000,E1 282.771} C_DIS
LIN {X -0.230,Y -454.738,Z 1353.568,A 0.000,B 0.000,C 90.000,E1 282.299} C_DIS
LIN {X -0.150,Y -456.576,Z 1353.565,A 0.000,B 0.000,C 90.000,E1 281.771} C_DIS
LIN {X -0.064,Y -458.106,Z 1353.562,A 0.000,B 0.000,C 90.000,E1 281.243} C_DIS
LIN {X 0.032,Y -459.212,Z 1353.560,A 0.000,B 0.000,C 90.000,E1 280.715} C_DIS
LIN {X 0.053,Y -459.887,Z 1353.557,A 0.000,B 0.000,C 90.000,E1 280.197} C_DIS
LIN {X 0.163,Y -460.171,Z 1353.554,A 0.000,B 0.000,C 90.000,E1 279.670} C_DIS
LIN {X 0.200,Y -459.934,Z 1353.551,A 0.000,B 0.000,C 90.000,E1 279.151} C_DIS
LIN {X -0.143,Y -459.227,Z 1353.548,A 0.000,B 0.000,C 90.000,E1 278.681} C_DIS
LIN {X -0.104,Y -458.012,Z 1353.545,A 0.000,B 0.000,C 90.000,E1 278.163} C_DIS
LIN {X -0.067,Y -456.251,Z 1353.542,A 0.000,B 0.000,C 90.000,E1 277.644} C_DIS
LIN {X 0.225,Y -452.614,Z 1353.538,A 0.000,B 0.000,C 90.000,E1 276.834} C_DIS
LIN {X -0.216,Y -449.520,Z 1353.535,A 0.000,B 0.000,C 90.000,E1 276.372} C_DIS
LIN {X 0.219,Y -445.760,Z 1353.532,A 0.000,B 0.000,C 90.000,E1 275.796} C_DIS
LIN {X 0.188,Y -441.147,Z 1353.529,A 0.000,B 0.000,C 90.000,E1 275.277} C_DIS
LIN {X -0.189,Y -435.612,Z 1353.527,A 0.000,B 0.000,C 90.000,E1 274.816} C_DIS
LIN {X 0.165,Y -429.541,Z 1353.524,A 0.000,B 0.000,C 90.000,E1 274.302} C_DIS
LIN {X 0.118,Y -423.159,Z 1353.522,A 0.000,B 0.000,C 90.000,E1 273.898} C_DIS
LIN {X -0.011,Y -416.647,Z 1353.520,A 0.000,B 0.000,C 90.000,E1 273.555} C_DIS
LIN {X 0.167,Y -410.077,Z 1353.518,A 0.000,B 0.000,C 90.000,E1 273.212} C_DIS
LIN {X 0.190,Y -403.395,Z 1353.516,A 0.000,B 0.000,C 90.000,E1 272.922} C_DIS
LIN {X 0.009,Y -396.455,Z 1353.515,A 0.000,B 0.000,C 90.000,E1 272.694} C_DIS
LIN {X 0.060,Y -389.414,Z 1353.514,A 0.000,B 0.000,C 90.000,E1 272.465} C_DIS
LIN {X 0.143,Y -378.403,Z 1353.512,A 0.000,B 0.000,C 90.000,E1 272.178} C_DIS
LIN {X -0.053,Y -370.129,Z 1353.511,A 0.000,B 0.000,C 90.000,E1 272.064} C_DIS
LIN {X 0.072,Y -356.877,Z 1353.511,A 0.000,B 0.000,C 90.000,E1 271.892} C_DIS
LIN {X -0.083,Y -345.410,Z 1353.510,A 0.000,B 0.000,C 90.000,E1 271.835} C_DIS
LIN {X 0.153,Y -336.335,Z 1353.510,A 0.000,B 0.000,C 90.000,E1 271.776} C_DIS
LIN {X 0.052,Y -181.297,Z 1353.510,A 0.000,B 0.000,C 90.000,E1 271.776} C_DIS
LIN {X -0.059,Y -181.581,Z 1353.501,A 0.000,B 0.000,C 90.000,E1 270.286} C_DIS
LIN {X 0.081,Y -180.908,Z 1353.475,A 0.000,B 0.000,C 90.000,E1 265.527} C_DIS
LIN {X -0.041,Y -180.771,Z 1353.471,A 0.000,B 0.000,C 90.000,E1 264.723} C_DIS
LIN {X 0.030,Y -178.866,Z 1353.443,A 0.000,B 0.000,C 90.000,E1 259.634} C_DIS
LIN {X -0.069,Y -175.909,Z 1353.414,A 0.000,B 0.000,C 90.000,E1 254.574} C_DIS
LIN {X -0.012,Y -174.596,Z 1353.405,A 0.000,B 0.000,C 90.000,E1 252.851} C_DIS
LIN {X -0.086,Y -171.578,Z 1353.381,A 0.000,B 0.000,C 90.000,E1 248.592} C_DIS
LIN {X -0.097,Y -167.801,Z 1353.357,A 0.000,B 0.000,C 90.000,E1 244.280} C_DIS
LIN {X 0.070,Y -166.519,Z 1353.347,A 0.000,B 0.000,C 90.000,E1 242.487} C_DIS
LIN {X 0.057,Y -162.521,Z 1353.323,A 0.000,B 0.000,C 90.000,E1 238.122} C_DIS
LIN {X 0.028,Y -161.194,Z 1353.313,A 0.000,B 0.000,C 90.000,E1 236.373} C_DIS
LIN {X -0.069,Y -157.205,Z 1353.289,A 0.000,B 0.000,C 90.000,E1 231.984} C_DIS
LIN {X -0.046,Y -155.932,Z 1353.279,A 0.000,B 0.000,C 90.000,E1 230.194} C_DIS
LIN {X -0.086,Y -152.183,Z 1353.254,A 0.000,B 0.000,C 90.000,E1 225.729} C_DIS
LIN {X -0.064,Y -150.431,Z 1353.239,A 0.000,B 0.000,C 90.000,E1 223.014} C_DIS
LIN {X -0.036,Y -147.158,Z 1353.214,A 0.000,B 0.000,C 90.000,E1 218.463} C_DIS
LIN {X -0.069,Y -145.174,Z 1353.193,A 0.000,B 0.000,C 90.000,E1 214.818} C_DIS
LIN {X -0.033,Y -142.322,Z 1353.163,A 0.000,B 0.000,C 90.000,E1 209.283} C_DIS
LIN {X -0.039,Y -141.712,Z 1353.152,A 0.000,B 0.000,C 90.000,E1 207.436} C_DIS
LIN {X 0.009,Y -139.472,Z 1353.116,A 0.000,B 0.000,C 90.000,E1 200.918} C_DIS
LIN {X -0.068,Y -139.204,Z 1353.106,A 0.000,B 0.000,C 90.000,E1 199.087} C_DIS
LIN {X -0.011,Y -138.329,Z 1353.054,A 0.000,B 0.000,C 90.000,E1 189.726} C_DIS
LIN {X -0.008,Y -139.439,Z 1353.007,A 0.000,B 0.000,C 90.000,E1 181.318} C_DIS
LIN {X 0.072,Y -140.971,Z 1352.976,A 0.000,B 0.000,C 90.000,E1 175.698} C_DIS
LIN {X 0.023,Y -142.727,Z 1352.956,A 0.000,B 0.000,C 90.000,E1 172.008} C_DIS
LIN {X -0.020,Y -145.112,Z 1352.930,A 0.000,B 0.000,C 90.000,E1 167.409} C_DIS
LIN {X -0.025,Y -147.735,Z 1352.910,A 0.000,B 0.000,C 90.000,E1 163.740} C_DIS
LIN {X 0.057,Y -150.399,Z 1352.889,A 0.000,B 0.000,C 90.000,E1 160.061} C_DIS
LIN {X -0.068,Y -153.835,Z 1352.869,A 0.000,B 0.000,C 90.000,E1 156.485} C_DIS
LIN {X -0.009,Y -157.246,Z 1352.849,A 0.000,B 0.000,C 90.000,E1 152.871} C_DIS
LIN {X -0.071,Y -161.418,Z 1352.829,A 0.000,B 0.000,C 90.000,E1 149.331} C_DIS
LIN {X -0.060,Y -165.619,Z 1352.810,A 0.000,B 0.000,C 90.000,E1 145.801} C_DIS
LIN {X 0.060,Y -170.547,Z 1352.791,A 0.000,B 0.000,C 90.000,E1 142.271} C_DIS
LIN {X -0.032,Y -175.426,Z 1352.771,A 0.000,B 0.000,C 90.000,E1 138.852} C_DIS
LIN {X 0.085,Y -181.049,Z 1352.752,A 0.000,B 0.000,C 90.000,E1 135.405} C_DIS
LIN {X -0.049,Y -186.484,Z 1352.734,A 0.000,B 0.000,C 90.000,E1 132.081} C_DIS
LIN {X 0.019,Y -191.106,Z 1352.720,A 0.000,B 0.000,C 90.000,E1 129.564} C_DIS
LIN {X -0.061,Y -196.900,Z 1352.702,A 0.000,B 0.000,C 90.000,E1 126.297} C_DIS
LIN {X 0.053,Y -199.193,Z 1352.695,A 0.000,B 0.000,C 90.000,E1 125.105} C_DIS
LIN {X 0.042,Y -308.822,Z 1352.695,A 0.000,B 0.000,C 90.000,E1 125.105} C_DIS
LIN {X -0.079,Y -310.539,Z 1352.695,A 0.000,B 0.000,C 90.000,E1 125.105} C_DIS
LIN {X -0.153,Y -315.486,Z 1352.694,A 0.000,B 0.000,C 90.000,E1 124.898} C_DIS
LIN {X -0.047,Y -318.093,Z 1352.693,A 0.000,B 0.000,C 90.000,E1 124.659} C_DIS
LIN {X -0.208,Y -321.866,Z 1352.690,A 0.000,B 0.000,C 90.000,E1 124.199} C_DIS
LIN {X 0.046,Y -323.579,Z 1352.688,A 0.000,B 0.000,C 90.000,E1 123.833} C_DIS
LIN {X -0.057,Y -326.012,Z 1352.684,A 0.000,B 0.000,C 90.000,E1 123.214} C_DIS
LIN {X -0.069,Y -336.482,Z 1352.669,A 0.000,B 0.000,C 90.000,E1 120.384} C_DIS
LIN {X 0.022,Y -348.294,Z 1352.653,A 0.000,B 0.000,C 90.000,E1 117.590} C_DIS
LIN {X -0.179,Y -361.555,Z 1352.638,A 0.000,B 0.000,C 90.000,E1 114.899} C_DIS
LIN {X -0.086,Y -374.650,Z 1352.625,A 0.000,B 0.000,C 90.000,E1 112.514} C_DIS
LIN {X 0.049,Y -389.068,Z 1352.612,A 0.000,B 0.000,C 90.000,E1 110.174} C_DIS
LIN {X -0.094,Y -404.914,Z 1352.599,A 0.000,B 0.000,C 90.000,E1 107.928} C_DIS
LIN {X -0.102,Y -422.295,Z 1352.587,A 0.000,B 0.000,C 90.000,E1 105.717} C_DIS
LIN {X 0.112,Y -441.330,Z 1352.575,A 0.000,B 0.000,C 90.000,E1 103.536} C_DIS
LIN {X -0.023,Y -461.374,Z 1352.564,A 0.000,B 0.000,C 90.000,E1 101.535} C_DIS
LIN {X -0.026,Y -479.348,Z 1352.555,A 0.000,B 0.000,C 90.000,E1 99.905} C_DIS
LIN {X 0.067,Y -481.739,Z 1352.554,A 0.000,B 0.000,C 90.000,E1 99.670} C_DIS
LIN {X -0.017,Y -483.629,Z 1352.552,A 0.000,B 0.000,C 90.000,E1 99.443} C_DIS
LIN {X -0.022,Y -485.065,Z 1352.551,A 0.000,B 0.000,C 90.000,E1 99.208} C_DIS
LIN {X 0.161,Y -487.024,Z 1352.548,A 0.000,B 0.000,C 90.000,E1 98.690} C_DIS
LIN {X -0.058,Y -487.847,Z 1352.546,A 0.000,B 0.000,C 90.000,E1 98.219} C_DIS
LIN {X 0.145,Y -487.680,Z 1352.543,A 0.000,B 0.000,C 90.000,E1 97.701} C_DIS
LIN {X -0.129,Y -486.498,Z 1352.540,A 0.000,B 0.000,C 90.000,E1 97.239} C_DIS
LIN {X 0.246,Y -485.471,Z 1352.539,A 0.000,B 0.000,C 90.000,E1 96.947} C_DIS
LIN {X 0.079,Y -484.085,Z 1352.537,A 0.000,B 0.000,C 90.000,E1 96.720} C_DIS
LIN {X -0.217,Y -469.973,Z 1352.526,A 0.000,B 0.000,C 90.000,E1 94.759} C_DIS
LIN {X -0.014,Y -460.069,Z 1352.518,A 0.000,B 0.000,C 90.000,E1 93.212} C_DIS
LIN {X -0.045,Y -443.501,Z 1352.503,A 0.000,B 0.000,C 90.000,E1 90.630} C_DIS
LIN {X -0.106,Y -428.578,Z 1352.489,A 0.000,B 0.000,C 90.000,E1 87.993} C_DIS
LIN {X 0.068,Y -416.878,Z 1352.477,A 0.000,B 0.000,C 90.000,E1 85.812} C_DIS
LIN {X -0.074,Y -406.541,Z 1352.466,A 0.000,B 0.000,C 90.000,E1 83.913} C_DIS
LIN {X 0.018,Y -395.954,Z 1352.455,A 0.000,B 0.000,C 90.000,E1 81.951} C_DIS
LIN {X -0.112,Y -386.656,Z 1352.446,A 0.000,B 0.000,C 90.000,E1 80.274} C_DIS
LIN {X 0.099,Y -377.194,Z 1352.436,A 0.000,B 0.000,C 90.000,E1 78.522} C_DIS
LIN {X 0.130,Y -367.443,Z 1352.427,A 0.000,B 0.000,C 90.000,E1 76.769} C_DIS
LIN {X 0.103,Y -355.908,Z 1352.415,A 0.000,B 0.000,C 90.000,E1 74.700} C_DIS
LIN {X 0.015,Y -345.988,Z 1352.405,A 0.000,B 0.000,C 90.000,E1 72.906} C_DIS
LIN {X -0.141,Y -336.004,Z 1352.395,A 0.000,B 0.000,C 90.000,E1 71.094} C_DIS
LIN {X -0.123,Y -322.846,Z 1352.381,A 0.000,B 0.000,C 90.000,E1 68.592} C_DIS
LIN {X -0.041,Y -305.771,Z 1352.361,A 0.000,B 0.000,C 90.000,E1 65.049} C_DIS
LIN {X -0.025,Y -297.310,Z 1352.350,A 0.000,B 0.000,C 90.000,E1 63.076} C_DIS
LIN {X 0.081,Y -287.249,Z 1352.336,A 0.000,B 0.000,C 90.000,E1 60.383} C_DIS
LIN {X 0.093,Y -278.482,Z 1352.320,A 0.000,B 0.000,C 90.000,E1 57.661} C_DIS
LIN {X 0.120,Y -270.521,Z 1352.305,A 0.000,B 0.000,C 90.000,E1 54.895} C_DIS
LIN {X 0.046,Y -262.954,Z 1352.290,A 0.000,B 0.000,C 90.000,E1 52.110} C_DIS
LIN {X -0.021,Y -253.936,Z 1352.270,A 0.000,B 0.000,C 90.000,E1 48.566} C_DIS
LIN {X 0.092,Y -245.445,Z 1352.250,A 0.000,B 0.000,C 90.000,E1 44.919} C_DIS
LIN {X 0.123,Y -237.748,Z 1352.229,A 0.000,B 0.000,C 90.000,E1 41.229} C_DIS
LIN {X -0.012,Y -230.837,Z 1352.208,A 0.000,B 0.000,C 90.000,E1 37.523} C_DIS
LIN {X 0.092,Y -224.762,Z 1352.187,A 0.000,B 0.000,C 90.000,E1 33.706} C_DIS
LIN {X 0.075,Y -219.679,Z 1352.166,A 0.000,B 0.000,C 90.000,E1 29.873} C_DIS
LIN {X 0.109,Y -214.936,Z 1352.140,A 0.000,B 0.000,C 90.000,E1 25.207} C_DIS
LIN {X -0.072,Y -211.440,Z 1352.114,A 0.000,B 0.000,C 90.000,E1 20.556} C_DIS
LIN {X -0.103,Y -208.978,Z 1352.092,A 0.000,B 0.000,C 90.000,E1 16.622} C_DIS
LIN {X -0.058,Y -206.670,Z 1352.070,A 0.000,B 0.000,C 90.000,E1 12.647} C_DIS
LIN {X 0.009,Y -204.960,Z 1352.052,A 0.000,B 0.000,C 90.000,E1 9.443} C_DIS
LIN {X -0.019,Y -203.042,Z 1352.030,A 0.000,B 0.000,C 90.000,E1 5.454} C_DIS
LIN {X -0.037,Y -201.035,Z 1351.997,A 0.000,B 0.000,C 90.000,E1 359.542} C_DIS
LIN {X -0.099,Y -200.374,Z 1351.962,A 0.000,B 0.000,C 90.000,E1 353.109} C_DIS
LIN {X -0.095,Y -202.199,Z 1351.917,A 0.000,B 0.000,C 90.000,E1 345.046} C_DIS
LIN {X 0.052,Y -205.484,Z 1351.886,A 0.000,B 0.000,C 90.000,E1 339.390} C_DIS
LIN {X -0.135,Y -209.823,Z 1351.859,A 0.000,B 0.000,C 90.000,E1 334.665} C_DIS
LIN {X 0.061,Y -214.610,Z 1351.837,A 0.000,B 0.000,C 90.000,E1 330.667} C_DIS
LIN {X -0.019,Y -220.585,Z 1351.815,A 0.000,B 0.000,C 90.000,E1 326.786} C_DIS
LIN {X 0.026,Y -227.683,Z 1351.794,A 0.000,B 0.000,C 90.000,E1 322.924} C_DIS
LIN {X -0.070,Y -234.213,Z 1351.777,A 0.000,B 0.000,C 90.000,E1 319.908} C_DIS
LIN {X -0.051,Y -241.535,Z 1351.760,A 0.000,B 0.000,C 90.000,E1 316.905} C_DIS
LIN {X -0.015,Y -250.726,Z 1351.742,A 0.000,B 0.000,C 90.000,E1 313.581} C_DIS
LIN {X -0.107,Y -258.883,Z 1351.728,A 0.000,B 0.000,C 90.000,E1 311.067} C_DIS
LIN {X 0.038,Y -268.067,Z 1351.714,A 0.000,B 0.000,C 90.000,E1 308.543} C_DIS
LIN {X 0.004,Y -279.900,Z 1351.699,A 0.000,B 0.000,C 90.000,E1 305.758} C_DIS
LIN {X -0.007,Y -289.783,Z 1351.687,A 0.000,B 0.000,C 90.000,E1 303.706} C_DIS
LIN {X 0.084,Y -299.124,Z 1351.678,A 0.000,B 0.000,C 90.000,E1 302.005} C_DIS
LIN {X 0.146,Y -307.318,Z 1351.671,A 0.000,B 0.000,C 90.000,E1 300.669} C_DIS
LIN {X -0.116,Y -316.402,Z 1351.663,A 0.000,B 0.000,C 90.000,E1 299.411} C_DIS
LIN {X 0.104,Y -328.949,Z 1351.654,A 0.000,B 0.000,C 90.000,E1 297.769} C_DIS
LIN {X -0.044,Y -347.483,Z 1351.642,A 0.000,B 0.000,C 90.000,E1 295.643} C_DIS
LIN {X -0.186,Y -363.393,Z 1351.633,A 0.000,B 0.000,C 90.000,E1 293.898} C_DIS
LIN {X 0.023,Y -376.369,Z 1351.625,A 0.000,B 0.000,C 90.000,E1 292.408} C_DIS
LIN {X -0.066,Y -388.860,Z 1351.616,A 0.000,B 0.000,C 90.000,E1 290.972} C_DIS
LIN {X -0.077,Y -403.575,Z 1351.607,A 0.000,B 0.000,C 90.000,E1 289.268} C_DIS
LIN {X 0.059,Y -418.280,Z 1351.598,A 0.000,B 0.000,C 90.000,E1 287.583} C_DIS
LIN {X 0.032,Y -427.656,Z 1351.592,A 0.000,B 0.000,C 90.000,E1 286.496} C_DIS
LIN {X 0.234,Y -434.255,Z 1351.587,A 0.000,B 0.000,C 90.000,E1 285.662} C_DIS
LIN {X -0.045,Y -440.286,Z 1351.583,A 0.000,B 0.000,C 90.000,E1 284.898} C_DIS
LIN {X -0.156,Y -445.601,Z 1351.578,A 0.000,B 0.000,C 90.000,E1 284.120} C_DIS
LIN {X 0.099,Y -450.097,Z 1351.574,A 0.000,B 0.000,C 90.000,E1 283.300} C_DIS
LIN {X -0.035,Y -453.798,Z 1351.570,A 0.000,B 0.000,C 90.000,E1 282.535} C_DIS
LIN {X -0.142,Y -456.777,Z 1351.565,A 0.000,B 0.000,C 90.000,E1 281.771} C_DIS
LIN {X -0.054,Y -458.303,Z 1351.562,A 0.000,B 0.000,C 90.000,E1 281.243} C_DIS
LIN {X 0.042,Y -459.436,Z 1351.560,A 0.000,B 0.000,C 90.000,E1 280.715} C_DIS
LIN {X 0.065,Y -460.126,Z 1351.557,A 0.000,B 0.000,C 90.000,E1 280.197} C_DIS
LIN {X 0.177,Y -460.400,Z 1351.554,A 0.000,B 0.000,C 90.000,E1 279.670} C_DIS
LIN {X -0.240,Y -460.203,Z 1351.551,A 0.000,B 0.000,C 90.000,E1 279.208} C_DIS
LIN {X -0.127,Y -459.522,Z 1351.548,A 0.000,B 0.000,C 90.000,E1 278.681} C_DIS
LIN {X -0.087,Y -458.323,Z 1351.545,A 0.000,B 0.000,C 90.000,E1 278.163} C_DIS
LIN {X -0.048,Y -456.604,Z 1351.542,A 0.000,B 0.000,C 90.000,E1 277.644} C_DIS
LIN {X -0.014,Y -454.308,Z 1351.540,A 0.000,B 0.000,C 90.000,E1 277.125} C_DIS
LIN {X 0.004,Y -451.581,Z 1351.537,A 0.000,B 0.000,C 90.000,E1 276.606} C_DIS
LIN {X 0.008,Y -448.188,Z 1351.534,A 0.000,B 0.000,C 90.000,E1 276.087} C_DIS
LIN {X -0.005,Y -444.125,Z 1351.531,A 0.000,B 0.000,C 90.000,E1 275.568} C_DIS
LIN {X 0.217,Y -441.760,Z 1351.529,A 0.000,B 0.000,C 90.000,E1 275.277} C_DIS
LIN {X -0.165,Y -436.275,Z 1351.527,A 0.000,B 0.000,C 90.000,E1 274.816} C_DIS
LIN {X 0.167,Y -430.242,Z 1351.524,A 0.000,B 0.000,C 90.000,E1 274.302} C_DIS
LIN {X 0.091,Y -423.911,Z 1351.522,A 0.000,B 0.000,C 90.000,E1 273.898} C_DIS
LIN {X -0.079,Y -417.357,Z 1351.520,A 0.000,B 0.000,C 90.000,E1 273.555} C_DIS
LIN {X 0.057,Y -410.784,Z 1351.518,A 0.000,B 0.000,C 90.000,E1 273.212} C_DIS
LIN {X 0.052,Y -404.086,Z 1351.516,A 0.000,B 0.000,C 90.000,E1 272.922} C_DIS
LIN {X -0.170,Y -393.561,Z 1351.514,A 0.000,B 0.000,C 90.000,E1 272.579} C_DIS
LIN {X -0.039,Y -386.243,Z 1351.513,A 0.000,B 0.000,C 90.000,E1 272.350} C_DIS
LIN {X -0.128,Y -375.367,Z 1351.512,A 0.000,B 0.000,C 90.000,E1 272.121} C_DIS
LIN {X 0.168,Y -367.010,Z 1351.511,A 0.000,B 0.000,C 90.000,E1 271.949} C_DIS
LIN {X -0.098,Y -357.704,Z 1351.510,A 0.000,B 0.000,C 90.000,E1 271.892} C_DIS
LIN {X 0.114,Y -344.848,Z 1351.510,A 0.000,B 0.000,C 90.000,E1 271.776} C_DIS
LIN {X 0.057,Y -341.913,Z 1351.510,A 0.000,B 0.000,C 90.000,E1 271.776} C_DIS
LIN {X 0.000,Y -181.300,Z 1351.510,A 0.000,B 0.000,C 90.000,E1 271.776} C_DIS
LIN {X 0.044,Y -181.581,Z 1351.501,A 0.000,B 0.000,C 90.000,E1 270.229} C_DIS
LIN {X 0.003,Y -180.907,Z 1351.475,A 0.000,B 0.000,C 90.000,E1 265.527} C_DIS
LIN {X 0.060,Y -180.761,Z 1351.470,A 0.000,B 0.000,C 90.000,E1 264.666} C_DIS
LIN {X -0.048,Y -178.855,Z 1351.442,A 0.000,B 0.000,C 90.000,E1 259.634} C_DIS
LIN {X 0.023,Y -175.898,Z 1351.414,A 0.000,B 0.000,C 90.000,E1 254.519} C_DIS
LIN {X -0.038,Y -174.575,Z 1351.405,A 0.000,B 0.000,C 90.000,E1 252.834} C_DIS
LIN {X -0.002,Y -171.559,Z 1351.381,A 0.000,B 0.000,C 90.000,E1 248.539} C_DIS
LIN {X 0.053,Y -167.782,Z 1351.357,A 0.000,B 0.000,C 90.000,E1 244.204} C_DIS
LIN {X -0.005,Y -166.495,Z 1351.347,A 0.000,B 0.000,C 90.000,E1 242.487} C_DIS
LIN {X -0.010,Y -163.206,Z 1351.328,A 0.000,B 0.000,C 90.000,E1 238.997} C_DIS
LIN {X -0.045,Y -161.169,Z 1351.313,A 0.000,B 0.000,C 90.000,E1 236.373} C_DIS
LIN {X 0.079,Y -157.184,Z 1351.289,A 0.000,B 0.000,C 90.000,E1 231.904} C_DIS
LIN {X 0.002,Y -155.914,Z 1351.279,A 0.000,B 0.000,C 90.000,E1 230.150} C_DIS
LIN {X 0.059,Y -152.164,Z 1351.254,A 0.000,B 0.000,C 90.000,E1 225.648} C_DIS
LIN {X -0.032,Y -150.413,Z 1351.239,A 0.000,B 0.000,C 90.000,E1 222.975} C_DIS
LIN {X 0.010,Y -147.142,Z 1351.214,A 0.000,B 0.000,C 90.000,E1 218.418} C_DIS
LIN {X 0.006,Y -145.701,Z 1351.198,A 0.000,B 0.000,C 90.000,E1 215.678} C_DIS
LIN {X 0.015,Y -143.084,Z 1351.173,A 0.000,B 0.000,C 90.000,E1 211.082} C_DIS
LIN {X 0.019,Y -141.701,Z 1351.152,A 0.000,B 0.000,C 90.000,E1 207.385} C_DIS
LIN {X -0.057,Y -139.467,Z 1351.116,A 0.000,B 0.000,C 90.000,E1 200.918} C_DIS
LIN {X -0.004,Y -139.200,Z 1351.106,A 0.000,B 0.000,C 90.000,E1 199.033} C_DIS
LIN {X 0.059,Y -138.327,Z 1351.054,A 0.000,B 0.000,C 90.000,E1 189.670} C_DIS
LIN {X 0.064,Y -139.444,Z 1351.007,A 0.000,B 0.000,C 90.000,E1 181.260} C_DIS
LIN {X 0.005,Y -140.983,Z 1350.976,A 0.000,B 0.000,C 90.000,E1 175.698} C_DIS
LIN {X -0.045,Y -142.738,Z 1350.955,A 0.000,B 0.000,C 90.000,E1 172.008} C_DIS
LIN {X 0.053,Y -145.129,Z 1350.930,A 0.000,B 0.000,C 90.000,E1 167.353} C_DIS
LIN {X 0.047,Y -147.753,Z 1350.909,A 0.000,B 0.000,C 90.000,E1 163.685} C_DIS
LIN {X -0.014,Y -150.422,Z 1350.889,A 0.000,B 0.000,C 90.000,E1 160.061} C_DIS
LIN {X 0.001,Y -153.863,Z 1350.869,A 0.000,B 0.000,C 90.000,E1 156.433} C_DIS
LIN {X -0.083,Y -157.273,Z 1350.849,A 0.000,B 0.000,C 90.000,E1 152.871} C_DIS
LIN {X -0.005,Y -161.452,Z 1350.829,A 0.000,B 0.000,C 90.000,E1 149.282} C_DIS
LIN {X 0.002,Y -165.652,Z 1350.810,A 0.000,B 0.000,C 90.000,E1 145.754} C_DIS
LIN {X -0.017,Y -170.587,Z 1350.790,A 0.000,B 0.000,C 90.000,E1 142.271} C_DIS
LIN {X -0.110,Y -175.464,Z 1350.771,A 0.000,B 0.000,C 90.000,E1 138.852} C_DIS
LIN {X 0.006,Y -181.087,Z 1350.752,A 0.000,B 0.000,C 90.000,E1 135.405} C_DIS
LIN {X -0.004,Y -186.529,Z 1350.734,A 0.000,B 0.000,C 90.000,E1 132.043} C_DIS
LIN {X -0.063,Y -191.146,Z 1350.720,A 0.000,B 0.000,C 90.000,E1 129.564} C_DIS
LIN {X 0.015,Y -196.947,Z 1350.701,A 0.000,B 0.000,C 90.000,E1 126.251} C_DIS
LIN {X 0.062,Y -199.188,Z 1350.695,A 0.000,B 0.000,C 90.000,E1 125.105} C_DIS
LIN {X 0.060,Y -308.424,Z 1350.695,A 0.000,B 0.000,C 90.000,E1 125.105} C_DIS
LIN {X -0.208,Y -311.523,Z 1350.695,A 0.000,B 0.000,C 90.000,E1 125.105} C_DIS
LIN {X 0.155,Y -315.823,Z 1350.694,A 0.000,B 0.000,C 90.000,E1 124.818} C_DIS
LIN {X 0.082,Y -318.321,Z 1350.692,A 0.000,B 0.000,C 90.000,E1 124.612} C_DIS
LIN {X 0.006,Y -322.097,Z 1350.690,A 0.000,B 0.000,C 90.000,E1 124.119} C_DIS
LIN {X 0.082,Y -323.752,Z 1350.688,A 0.000,B 0.000,C 90.000,E1 123.785} C_DIS
LIN {X -0.018,Y -326.132,Z 1350.684,A 0.000,B 0.000,C 90.000,E1 123.166} C_DIS
LIN {X -0.016,Y -336.621,Z 1350.668,A 0.000,B 0.000,C 90.000,E1 120.335} C_DIS
LIN {X -0.059,Y -348.453,Z 1350.653,A 0.000,B 0.000,C 90.000,E1 117.564} C_DIS
LIN {X 0.055,Y -361.735,Z 1350.638,A 0.000,B 0.000,C 90.000,E1 114.823} C_DIS
LIN {X 0.009,Y -374.850,Z 1350.625,A 0.000,B 0.000,C 90.000,E1 112.461} C_DIS
LIN {X 0.160,Y -389.292,Z 1350.612,A 0.000,B 0.000,C 90.000,E1 110.120} C_DIS
LIN {X 0.031,Y -405.161,Z 1350.599,A 0.000,B 0.000,C 90.000,E1 107.873} C_DIS
LIN {X 0.039,Y -422.567,Z 1350.587,A 0.000,B 0.000,C 90.000,E1 105.662} C_DIS
LIN {X -0.155,Y -441.627,Z 1350.575,A 0.000,B 0.000,C 90.000,E1 103.536} C_DIS
LIN {X 0.173,Y -461.680,Z 1350.564,A 0.000,B 0.000,C 90.000,E1 101.478} C_DIS
LIN {X 0.198,Y -479.661,Z 1350.555,A 0.000,B 0.000,C 90.000,E1 99.849} C_DIS
LIN {X -0.181,Y -481.948,Z 1350.554,A 0.000,B 0.000,C 90.000,E1 99.670} C_DIS
LIN {X 0.238,Y -483.793,Z 1350.552,A 0.000,B 0.000,C 90.000,E1 99.378} C_DIS
LIN {X 0.103,Y -485.188,Z 1350.551,A 0.000,B 0.000,C 90.000,E1 99.151} C_DIS
LIN {X -0.120,Y -487.016,Z 1350.548,A 0.000,B 0.000,C 90.000,E1 98.681} C_DIS
LIN {X 0.070,Y -487.736,Z 1350.545,A 0.000,B 0.000,C 90.000,E1 98.163} C_DIS
LIN {X -0.209,Y -487.468,Z 1350.543,A 0.000,B 0.000,C 90.000,E1 97.701} C_DIS
LIN {X 0.000,Y -486.175,Z 1350.540,A 0.000,B 0.000,C 90.000,E1 97.182} C_DIS
LIN {X -0.108,Y -485.081,Z 1350.539,A 0.000,B 0.000,C 90.000,E1 96.947} C_DIS
LIN {X 0.206,Y -483.611,Z 1350.537,A 0.000,B 0.000,C 90.000,E1 96.663} C_DIS
LIN {X 0.048,Y -471.140,Z 1350.527,A 0.000,B 0.000,C 90.000,E1 94.935} C_DIS
LIN {X 0.090,Y -459.553,Z 1350.518,A 0.000,B 0.000,C 90.000,E1 93.154} C_DIS
LIN {X 0.041,Y -442.993,Z 1350.503,A 0.000,B 0.000,C 90.000,E1 90.573} C_DIS
LIN {X -0.037,Y -428.103,Z 1350.489,A 0.000,B 0.000,C 90.000,E1 87.936} C_DIS
LIN {X 0.124,Y -416.437,Z 1350.477,A 0.000,B 0.000,C 90.000,E1 85.755} C_DIS
LIN {X -0.031,Y -406.096,Z 1350.466,A 0.000,B 0.000,C 90.000,E1 83.856} C_DIS
LIN {X 0.049,Y -395.499,Z 1350.455,A 0.000,B 0.000,C 90.000,E1 81.894} C_DIS
LIN {X -0.026,Y -386.229,Z 1350.446,A 0.000,B 0.000,C 90.000,E1 80.208} C_DIS
LIN {X 0.124,Y -375.126,Z 1350.434,A 0.000,B 0.000,C 90.000,E1 78.173} C_DIS
LIN {X -0.157,Y -365.344,Z 1350.425,A 0.000,B 0.000,C 90.000,E1 76.464} C_DIS
LIN {X 0.135,Y -353.807,Z 1350.413,A 0.000,B 0.000,C 90.000,E1 74.338} C_DIS
LIN {X 0.011,Y -343.881,Z 1350.403,A 0.000,B 0.000,C 90.000,E1 72.543} C_DIS
LIN {X 0.119,Y -332.209,Z 1350.391,A 0.000,B 0.000,C 90.000,E1 70.369} C_DIS
LIN {X 0.148,Y -319.182,Z 1350.377,A 0.000,B 0.000,C 90.000,E1 67.847} C_DIS
LIN {X -0.048,Y -302.469,Z 1350.357,A 0.000,B 0.000,C 90.000,E1 64.332} C_DIS
LIN {X -0.088,Y -293.041,Z 1350.344,A 0.000,B 0.000,C 90.000,E1 62.025} C_DIS
LIN {X -0.050,Y -284.627,Z 1350.331,A 0.000,B 0.000,C 90.000,E1 59.665} C_DIS
LIN {X 0.100,Y -274.201,Z 1350.312,A 0.000,B 0.000,C 90.000,E1 56.215} C_DIS
LIN {X -0.051,Y -264.591,Z 1350.293,A 0.000,B 0.000,C 90.000,E1 52.763} C_DIS
LIN {X -0.060,Y -255.529,Z 1350.273,A 0.000,B 0.000,C 90.000,E1 49.218} C_DIS
LIN {X 0.120,Y -246.960,Z 1350.253,A 0.000,B 0.000,C 90.000,E1 45.567} C_DIS
LIN {X 0.021,Y -239.129,Z 1350.233,A 0.000,B 0.000,C 90.000,E1 41.919} C_DIS
LIN {X 0.080,Y -232.086,Z 1350.212,A 0.000,B 0.000,C 90.000,E1 38.177} C_DIS
LIN {X 0.039,Y -225.841,Z 1350.191,A 0.000,B 0.000,C 90.000,E1 34.405} C_DIS
LIN {X -0.016,Y -220.629,Z 1350.170,A 0.000,B 0.000,C 90.000,E1 30.590} C_DIS
LIN {X 0.055,Y -215.648,Z 1350.144,A 0.000,B 0.000,C 90.000,E1 25.924} C_DIS
LIN {X 0.069,Y -211.982,Z 1350.118,A 0.000,B 0.000,C 90.000,E1 21.227} C_DIS
LIN {X -0.082,Y -209.450,Z 1350.096,A 0.000,B 0.000,C 90.000,E1 17.330} C_DIS
LIN {X 0.081,Y -207.549,Z 1350.079,A 0.000,B 0.000,C 90.000,E1 14.120} C_DIS
LIN {X 0.046,Y -205.761,Z 1350.061,A 0.000,B 0.000,C 90.000,E1 10.950} C_DIS
LIN {X 0.090,Y -203.681,Z 1350.039,A 0.000,B 0.000,C 90.000,E1 6.947} C_DIS
LIN {X -0.063,Y -201.467,Z 1350.008,A 0.000,B 0.000,C 90.000,E1 1.375} C_DIS
LIN {X -0.080,Y -200.475,Z 1349.979,A 0.000,B 0.000,C 90.000,E1 356.331} C_DIS
LIN {X -0.018,Y -200.743,Z 1349.944,A 0.000,B 0.000,C 90.000,E1 349.859} C_DIS
LIN {X -0.070,Y -203.028,Z 1349.908,A 0.000,B 0.000,C 90.000,E1 343.433} C_DIS
LIN {X 0.057,Y -206.866,Z 1349.877,A 0.000,B 0.000,C 90.000,E1 337.794} C_DIS
LIN {X -0.020,Y -210.840,Z 1349.855,A 0.000,B 0.000,C 90.000,E1 333.845} C_DIS
LIN {X -0.063,Y -215.858,Z 1349.833,A 0.000,B 0.000,C 90.000,E1 329.921} C_DIS
LIN {X 0.020,Y -222.079,Z 1349.811,A 0.000,B 0.000,C 90.000,E1 326.008} C_DIS
LIN {X -0.065,Y -229.413,Z 1349.790,A 0.000,B 0.000,C 90.000,E1 322.190} C_DIS
LIN {X 0.034,Y -236.118,Z 1349.773,A 0.000,B 0.000,C 90.000,E1 319.138} C_DIS
LIN {X -0.089,Y -244.597,Z 1349.754,A 0.000,B 0.000,C 90.000,E1 315.810} C_DIS
LIN {X -0.139,Y -254.203,Z 1349.736,A 0.000,B 0.000,C 90.000,E1 312.528} C_DIS
LIN {X -0.090,Y -264.105,Z 1349.720,A 0.000,B 0.000,C 90.000,E1 309.644} C_DIS
LIN {X 0.010,Y -273.911,Z 1349.706,A 0.000,B 0.000,C 90.000,E1 307.156} C_DIS
LIN {X -0.003,Y -284.833,Z 1349.693,A 0.000,B 0.000,C 90.000,E1 304.739} C_DIS
LIN {X 0.011,Y -293.514,Z 1349.684,A 0.000,B 0.000,C 90.000,E1 303.038} C_DIS
LIN {X -0.072,Y -305.295,Z 1349.672,A 0.000,B 0.000,C 90.000,E1 301.052} C_DIS
LIN {X -0.093,Y -314.146,Z 1349.665,A 0.000,B 0.000,C 90.000,E1 299.745} C_DIS
LIN {X 0.112,Y -326.376,Z 1349.656,A 0.000,B 0.000,C 90.000,E1 298.103} C_DIS
LIN {X -0.089,Y -347.448,Z 1349.642,A 0.000,B 0.000,C 90.000,E1 295.668} C_DIS
LIN {X -0.095,Y -363.358,Z 1349.633,A 0.000,B 0.000,C 90.000,E1 293.898} C_DIS
LIN {X -0.214,Y -376.298,Z 1349.625,A 0.000,B 0.000,C 90.000,E1 292.461} C_DIS
LIN {X 0.050,Y -388.800,Z 1349.617,A 0.000,B 0.000,C 90.000,E1 290.972} C_DIS
LIN {X 0.043,Y -403.481,Z 1349.607,A 0.000,B 0.000,C 90.000,E1 289.268} C_DIS
LIN {X -0.217,Y -418.199,Z 1349.598,A 0.000,B 0.000,C 90.000,E1 287.638} C_DIS
LIN {X 0.156,Y -427.596,Z 1349.592,A 0.000,B 0.000,C 90.000,E1 286.496} C_DIS
LIN {X -0.059,Y -434.204,Z 1349.587,A 0.000,B 0.000,C 90.000,E1 285.717} C_DIS
LIN {X 0.081,Y -440.231,Z 1349.583,A 0.000,B 0.000,C 90.000,E1 284.898} C_DIS
LIN {X -0.029,Y -445.568,Z 1349.578,A 0.000,B 0.000,C 90.000,E1 284.120} C_DIS
LIN {X -0.210,Y -450.109,Z 1349.574,A 0.000,B 0.000,C 90.000,E1 283.355} C_DIS
LIN {X 0.095,Y -453.838,Z 1349.570,A 0.000,B 0.000,C 90.000,E1 282.535} C_DIS
LIN {X -0.011,Y -456.863,Z 1349.565,A 0.000,B 0.000,C 90.000,E1 281.771} C_DIS
LIN {X 0.077,Y -458.435,Z 1349.563,A 0.000,B 0.000,C 90.000,E1 281.243} C_DIS
LIN {X 0.090,Y -459.590,Z 1349.560,A 0.000,B 0.000,C 90.000,E1 280.725} C_DIS
LIN {X 0.199,Y -460.331,Z 1349.557,A 0.000,B 0.000,C 90.000,E1 280.197} C_DIS
LIN {X -0.143,Y -460.624,Z 1349.554,A 0.000,B 0.000,C 90.000,E1 279.726} C_DIS
LIN {X -0.104,Y -460.479,Z 1349.551,A 0.000,B 0.000,C 90.000,E1 279.208} C_DIS
LIN {X 0.008,Y -459.839,Z 1349.548,A 0.000,B 0.000,C 90.000,E1 278.681} C_DIS
LIN {X 0.050,Y -458.676,Z 1349.545,A 0.000,B 0.000,C 90.000,E1 278.163} C_DIS
LIN {X 0.091,Y -457.016,Z 1349.542,A 0.000,B 0.000,C 90.000,E1 277.644} C_DIS
LIN {X 0.126,Y -454.819,Z 1349.540,A 0.000,B 0.000,C 90.000,E1 277.125} C_DIS
LIN {X 0.146,Y -452.116,Z 1349.537,A 0.000,B 0.000,C 90.000,E1 276.606} C_DIS
LIN {X 0.152,Y -448.778,Z 1349.534,A 0.000,B 0.000,C 90.000,E1 276.087} C_DIS
LIN {X -0.054,Y -446.915,Z 1349.532,A 0.000,B 0.000,C 90.000,E1 275.853} C_DIS
LIN {X -0.076,Y -442.464,Z 1349.530,A 0.000,B 0.000,C 90.000,E1 275.334} C_DIS
LIN {X 0.107,Y -439.889,Z 1349.528,A 0.000,B 0.000,C 90.000,E1 275.049} C_DIS
LIN {X 0.157,Y -433.945,Z 1349.525,A 0.000,B 0.000,C 90.000,E1 274.531} C_DIS
LIN {X -0.193,Y -427.757,Z 1349.523,A 0.000,B 0.000,C 90.000,E1 274.131} C_DIS
LIN {X -0.110,Y -421.327,Z 1349.521,A 0.000,B 0.000,C 90.000,E1 273.726} C_DIS
LIN {X -0.126,Y -414.847,Z 1349.519,A 0.000,B 0.000,C 90.000,E1 273.383} C_DIS
LIN {X -0.041,Y -405.013,Z 1349.516,A 0.000,B 0.000,C 90.000,E1 272.922} C_DIS
LIN {X 0.146,Y -398.080,Z 1349.515,A 0.000,B 0.000,C 90.000,E1 272.636} C_DIS
LIN {X -0.117,Y -387.399,Z 1349.513,A 0.000,B 0.000,C 90.000,E1 272.350} C_DIS
LIN {X 0.123,Y -376.229,Z 1349.512,A 0.000,B 0.000,C 90.000,E1 272.064} C_DIS
LIN {X 0.026,Y -368.072,Z 1349.511,A 0.000,B 0.000,C 90.000,E1 271.949} C_DIS
LIN {X 0.108,Y -358.576,Z 1349.510,A 0.000,B 0.000,C 90.000,E1 271.835} C_DIS
LIN {X -0.029,Y -346.312,Z 1349.510,A 0.000,B 0.000,C 90.000,E1 271.776} C_DIS
LIN {X -0.084,Y -342.091,Z 1349.510,A 0.000,B 0.000,C 90.000,E1 271.776} C_DIS
LIN {X -0.074,Y -181.304,Z 1349.510,A 0.000,B 0.000,C 90.000,E1 271.776} C_DIS
LIN {X -0.029,Y -181.580,Z 1349.501,A 0.000,B 0.000,C 90.000,E1 270.229} C_DIS
LIN {X -0.070,Y -180.907,Z 1349.475,A 0.000,B 0.000,C 90.000,E1 265.527} C_DIS
LIN {X -0.013,Y -180.751,Z 1349.470,A 0.000,B 0.000,C 90.000,E1 264.666} C_DIS
LIN {X 0.055,Y -178.844,Z 1349.442,A 0.000,B 0.000,C 90.000,E1 259.577} C_DIS
LIN {X -0.049,Y -175.887,Z 1349.414,A 0.000,B 0.000,C 90.000,E1 254.519} C_DIS
LIN {X 0.057,Y -174.555,Z 1349.404,A 0.000,B 0.000,C 90.000,E1 252.779} C_DIS
LIN {X -0.073,Y -171.539,Z 1349.381,A 0.000,B 0.000,C 90.000,E1 248.539} C_DIS
LIN {X -0.017,Y -167.764,Z 1349.357,A 0.000,B 0.000,C 90.000,E1 244.204} C_DIS
LIN {X -0.075,Y -166.472,Z 1349.347,A 0.000,B 0.000,C 90.000,E1 242.487} C_DIS
LIN {X -0.078,Y -163.185,Z 1349.328,A 0.000,B 0.000,C 90.000,E1 238.997} C_DIS
LIN {X -0.024,Y -161.147,Z 1349.313,A 0.000,B 0.000,C 90.000,E1 236.342} C_DIS
LIN {X 0.012,Y -157.166,Z 1349.288,A 0.000,B 0.000,C 90.000,E1 231.904} C_DIS
LIN {X 0.035,Y -155.897,Z 1349.278,A 0.000,B 0.000,C 90.000,E1 230.114} C_DIS
LIN {X -0.007,Y -152.147,Z 1349.254,A 0.000,B 0.000,C 90.000,E1 225.648} C_DIS
LIN {X 0.013,Y -150.396,Z 1349.239,A 0.000,B 0.000,C 90.000,E1 222.933} C_DIS
LIN {X 0.036,Y -147.127,Z 1349.213,A 0.000,B 0.000,C 90.000,E1 218.382} C_DIS
LIN {X 0.027,Y -145.690,Z 1349.198,A 0.000,B 0.000,C 90.000,E1 215.644} C_DIS
LIN {X 0.024,Y -143.072,Z 1349.173,A 0.000,B 0.000,C 90.000,E1 211.052} C_DIS
LIN {X -0.044,Y -141.692,Z 1349.152,A 0.000,B 0.000,C 90.000,E1 207.385} C_DIS
LIN {X 0.010,Y -139.462,Z 1349.116,A 0.000,B 0.000,C 90.000,E1 200.865} C_DIS
LIN {X -0.066,Y -139.196,Z 1349.106,A 0.000,B 0.000,C 90.000,E1 199.033} C_DIS
LIN {X -0.003,Y -138.326,Z 1349.054,A 0.000,B 0.000,C 90.000,E1 189.670} C_DIS
LIN {X 0.002,Y -139.450,Z 1349.007,A 0.000,B 0.000,C 90.000,E1 181.260} C_DIS
LIN {X -0.058,Y -140.993,Z 1348.976,A 0.000,B 0.000,C 90.000,E1 175.698} C_DIS
LIN {X 0.032,Y -142.748,Z 1348.955,A 0.000,B 0.000,C 90.000,E1 171.951} C_DIS
LIN {X -0.011,Y -145.145,Z 1348.930,A 0.000,B 0.000,C 90.000,E1 167.353} C_DIS
LIN {X -0.018,Y -147.769,Z 1348.909,A 0.000,B 0.000,C 90.000,E1 163.685} C_DIS
LIN {X 0.061,Y -150.442,Z 1348.889,A 0.000,B 0.000,C 90.000,E1 160.007} C_DIS
LIN {X -0.004,Y -153.889,Z 1348.869,A 0.000,B 0.000,C 90.000,E1 156.410} C_DIS
LIN {X -0.010,Y -157.300,Z 1348.849,A 0.000,B 0.000,C 90.000,E1 152.820} C_DIS
LIN {X 0.009,Y -161.484,Z 1348.829,A 0.000,B 0.000,C 90.000,E1 149.253} C_DIS
LIN {X 0.025,Y -165.683,Z 1348.810,A 0.000,B 0.000,C 90.000,E1 145.722} C_DIS
LIN {X -0.088,Y -170.625,Z 1348.790,A 0.000,B 0.000,C 90.000,E1 142.271} C_DIS
LIN {X 0.066,Y -175.501,Z 1348.771,A 0.000,B 0.000,C 90.000,E1 138.771} C_DIS
LIN {X -0.068,Y -181.122,Z 1348.752,A 0.000,B 0.000,C 90.000,E1 135.405} C_DIS
LIN {X 0.059,Y -186.569,Z 1348.733,A 0.000,B 0.000,C 90.000,E1 132.000} C_DIS
LIN {X 0.009,Y -191.182,Z 1348.720,A 0.000,B 0.000,C 90.000,E1 129.519} C_DIS
LIN {X 0.055,Y -196.989,Z 1348.701,A 0.000,B 0.000,C 90.000,E1 126.217} C_DIS
LIN {X 0.045,Y -199.198,Z 1348.695,A 0.000,B 0.000,C 90.000,E1 125.105} C_DIS
LIN {X 0.023,Y -309.397,Z 1348.695,A 0.000,B 0.000,C 90.000,E1 125.105} C_DIS
LIN {X 0.186,Y -315.716,Z 1348.694,A 0.000,B 0.000,C 90.000,E1 124.818} C_DIS
LIN {X -0.043,Y -318.509,Z 1348.692,A 0.000,B 0.000,C 90.000,E1 124.612} C_DIS
LIN {X -0.140,Y -322.225,Z 1348.689,A 0.000,B 0.000,C 90.000,E1 124.119} C_DIS
LIN {X -0.065,Y -323.846,Z 1348.688,A 0.000,B 0.000,C 90.000,E1 123.785} C_DIS
LIN {X -0.070,Y -327.305,Z 1348.682,A 0.000,B 0.000,C 90.000,E1 122.832} C_DIS
LIN {X -0.029,Y -337.947,Z 1348.667,A 0.000,B 0.000,C 90.000,E1 120.001} C_DIS
LIN {X 0.109,Y -349.949,Z 1348.651,A 0.000,B 0.000,C 90.000,E1 117.206} C_DIS
LIN {X -0.039,Y -363.410,Z 1348.636,A 0.000,B 0.000,C 90.000,E1 114.515} C_DIS
LIN {X -0.041,Y -376.698,Z 1348.623,A 0.000,B 0.000,C 90.000,E1 112.153} C_DIS
LIN {X 0.153,Y -391.326,Z 1348.610,A 0.000,B 0.000,C 90.000,E1 109.812} C_DIS
LIN {X -0.053,Y -407.395,Z 1348.598,A 0.000,B 0.000,C 90.000,E1 107.583} C_DIS
LIN {X 0.017,Y -425.019,Z 1348.585,A 0.000,B 0.000,C 90.000,E1 105.371} C_DIS
LIN {X -0.076,Y -444.266,Z 1348.573,A 0.000,B 0.000,C 90.000,E1 103.244} C_DIS
LIN {X -0.012,Y -464.398,Z 1348.563,A 0.000,B 0.000,C 90.000,E1 101.243} C_DIS
LIN {X 0.041,Y -479.848,Z 1348.555,A 0.000,B 0.000,C 90.000,E1 99.849} C_DIS
LIN {X 0.137,Y -482.049,Z 1348.553,A 0.000,B 0.000,C 90.000,E1 99.613} C_DIS
LIN {X 0.035,Y -483.868,Z 1348.552,A 0.000,B 0.000,C 90.000,E1 99.378} C_DIS
LIN {X -0.146,Y -485.235,Z 1348.551,A 0.000,B 0.000,C 90.000,E1 99.151} C_DIS
LIN {X 0.111,Y -486.967,Z 1348.548,A 0.000,B 0.000,C 90.000,E1 98.624} C_DIS
LIN {X -0.180,Y -487.607,Z 1348.545,A 0.000,B 0.000,C 90.000,E1 98.163} C_DIS
LIN {X 0.024,Y -487.264,Z 1348.542,A 0.000,B 0.000,C 90.000,E1 97.644} C_DIS
LIN {X -0.251,Y -485.885,Z 1348.540,A 0.000,B 0.000,C 90.000,E1 97.182} C_DIS
LIN {X 0.122,Y -484.738,Z 1348.538,A 0.000,B 0.000,C 90.000,E1 96.891} C_DIS
LIN {X -0.044,Y -483.202,Z 1348.537,A 0.000,B 0.000,C 90.000,E1 96.663} C_DIS
LIN {X -0.203,Y -470.716,Z 1348.527,A 0.000,B 0.000,C 90.000,E1 94.935} C_DIS
LIN {X 0.048,Y -460.795,Z 1348.519,A 0.000,B 0.000,C 90.000,E1 93.383} C_DIS
LIN {X -0.216,Y -442.572,Z 1348.503,A 0.000,B 0.000,C 90.000,E1 90.573} C_DIS
LIN {X 0.131,Y -427.702,Z 1348.488,A 0.000,B 0.000,C 90.000,E1 87.879} C_DIS
LIN {X 0.146,Y -417.513,Z 1348.478,A 0.000,B 0.000,C 90.000,E1 85.988} C_DIS
LIN {X 0.009,Y -407.214,Z 1348.467,A 0.000,B 0.000,C 90.000,E1 84.090} C_DIS
LIN {X 0.078,Y -398.175,Z 1348.458,A 0.000,B 0.000,C 90.000,E1 82.413} C_DIS
LIN {X -0.012,Y -388.967,Z 1348.448,A 0.000,B 0.000,C 90.000,E1 80.735} C_DIS
LIN {X -0.178,Y -377.935,Z 1348.437,A 0.000,B 0.000,C 90.000,E1 78.757} C_DIS
LIN {X -0.045,Y -368.247,Z 1348.428,A 0.000,B 0.000,C 90.000,E1 76.992} C_DIS
LIN {X -0.125,Y -356.712,Z 1348.416,A 0.000,B 0.000,C 90.000,E1 74.936} C_DIS
LIN {X 0.141,Y -346.833,Z 1348.406,A 0.000,B 0.000,C 90.000,E1 73.087} C_DIS
LIN {X -0.011,Y -335.148,Z 1348.394,A 0.000,B 0.000,C 90.000,E1 70.967} C_DIS
LIN {X -0.015,Y -322.032,Z 1348.380,A 0.000,B 0.000,C 90.000,E1 68.465} C_DIS
LIN {X 0.038,Y -305.038,Z 1348.361,A 0.000,B 0.000,C 90.000,E1 64.921} C_DIS
LIN {X 0.043,Y -295.315,Z 1348.348,A 0.000,B 0.000,C 90.000,E1 62.615} C_DIS
LIN {X -0.040,Y -285.508,Z 1348.333,A 0.000,B 0.000,C 90.000,E1 59.950} C_DIS
LIN {X -0.115,Y -277.978,Z 1348.320,A 0.000,B 0.000,C 90.000,E1 57.582} C_DIS
LIN {X -0.078,Y -268.164,Z 1348.301,A 0.000,B 0.000,C 90.000,E1 54.116} C_DIS
LIN {X -0.043,Y -260.743,Z 1348.285,A 0.000,B 0.000,C 90.000,E1 51.295} C_DIS
LIN {X -0.010,Y -251.922,Z 1348.265,A 0.000,B 0.000,C 90.000,E1 47.715} C_DIS
LIN {X -0.134,Y -243.677,Z 1348.245,A 0.000,B 0.000,C 90.000,E1 44.109} C_DIS
LIN {X 0.019,Y -236.147,Z 1348.224,A 0.000,B 0.000,C 90.000,E1 40.378} C_DIS
LIN {X -0.126,Y -229.434,Z 1348.203,A 0.000,B 0.000,C 90.000,E1 36.664} C_DIS
LIN {X -0.003,Y -223.620,Z 1348.182,A 0.000,B 0.000,C 90.000,E1 32.832} C_DIS
LIN {X -0.054,Y -218.802,Z 1348.161,A 0.000,B 0.000,C 90.000,E1 28.999} C_DIS
LIN {X -0.053,Y -214.355,Z 1348.135,A 0.000,B 0.000,C 90.000,E1 24.335} C_DIS
LIN {X -0.098,Y -211.477,Z 1348.113,A 0.000,B 0.000,C 90.000,E1 20.429} C_DIS
LIN {X 0.068,Y -208.968,Z 1348.091,A 0.000,B 0.000,C 90.000,E1 16.441} C_DIS
LIN {X -0.031,Y -207.064,Z 1348.074,A 0.000,B 0.000,C 90.000,E1 13.300} C_DIS
LIN {X -0.115,Y -205.264,Z 1348.056,A 0.000,B 0.000,C 90.000,E1 10.141} C_DIS
LIN {X -0.106,Y -203.224,Z 1348.034,A 0.000,B 0.000,C 90.000,E1 6.144} C_DIS
LIN {X -0.036,Y -200.997,Z 1347.997,A 0.000,B 0.000,C 90.000,E1 359.542} C_DIS
LIN {X -0.099,Y -200.400,Z 1347.962,A 0.000,B 0.000,C 90.000,E1 353.109} C_DIS
LIN {X 0.003,Y -201.995,Z 1347.921,A 0.000,B 0.000,C 90.000,E1 345.825} C_DIS
LIN {X 0.069,Y -205.130,Z 1347.890,A 0.000,B 0.000,C 90.000,E1 340.188} C_DIS
LIN {X 0.063,Y -209.257,Z 1347.864,A 0.000,B 0.000,C 90.000,E1 335.409} C_DIS
LIN {X 0.054,Y -213.891,Z 1347.842,A 0.000,B 0.000,C 90.000,E1 331.463} C_DIS
LIN {X -0.050,Y -219.619,Z 1347.820,A 0.000,B 0.000,C 90.000,E1 327.582} C_DIS
LIN {X 0.023,Y -226.494,Z 1347.798,A 0.000,B 0.000,C 90.000,E1 323.703} C_DIS
LIN {X -0.008,Y -234.524,Z 1347.777,A 0.000,B 0.000,C 90.000,E1 319.908} C_DIS
LIN {X 0.022,Y -241.781,Z 1347.761,A 0.000,B 0.000,C 90.000,E1 316.905} C_DIS
LIN {X -0.113,Y -250.944,Z 1347.742,A 0.000,B 0.000,C 90.000,E1 313.623} C_DIS
LIN {X -0.016,Y -259.103,Z 1347.728,A 0.000,B 0.000,C 90.000,E1 311.067} C_DIS
LIN {X -0.072,Y -268.264,Z 1347.714,A 0.000,B 0.000,C 90.000,E1 308.588} C_DIS
LIN {X -0.054,Y -278.562,Z 1347.701,A 0.000,B 0.000,C 90.000,E1 306.137} C_DIS
LIN {X -0.024,Y -288.311,Z 1347.689,A 0.000,B 0.000,C 90.000,E1 304.072} C_DIS
LIN {X 0.054,Y -295.526,Z 1347.682,A 0.000,B 0.000,C 90.000,E1 302.704} C_DIS
LIN {X -0.009,Y -305.413,Z 1347.672,A 0.000,B 0.000,C 90.000,E1 301.052} C_DIS
LIN {X -0.027,Y -314.232,Z 1347.665,A 0.000,B 0.000,C 90.000,E1 299.745} C_DIS
LIN {X 0.154,Y -326.460,Z 1347.656,A 0.000,B 0.000,C 90.000,E1 298.103} C_DIS
LIN {X -0.050,Y -347.513,Z 1347.643,A 0.000,B 0.000,C 90.000,E1 295.668} C_DIS
LIN {X -0.077,Y -363.415,Z 1347.633,A 0.000,B 0.000,C 90.000,E1 293.898} C_DIS
LIN {X -0.199,Y -376.345,Z 1347.625,A 0.000,B 0.000,C 90.000,E1 292.461} C_DIS
LIN {X 0.066,Y -388.839,Z 1347.617,A 0.000,B 0.000,C 90.000,E1 290.972} C_DIS
LIN {X 0.065,Y -403.507,Z 1347.607,A 0.000,B 0.000,C 90.000,E1 289.268} C_DIS
LIN {X 0.097,Y -415.805,Z 1347.599,A 0.000,B 0.000,C 90.000,E1 287.873} C_DIS
LIN {X -0.084,Y -425.343,Z 1347.593,A 0.000,B 0.000,C 90.000,E1 286.804} C_DIS
LIN {X -0.034,Y -434.262,Z 1347.587,A 0.000,B 0.000,C 90.000,E1 285.717} C_DIS
LIN {X 0.106,Y -440.265,Z 1347.583,A 0.000,B 0.000,C 90.000,E1 284.898} C_DIS
LIN {X -0.002,Y -445.627,Z 1347.578,A 0.000,B 0.000,C 90.000,E1 284.120} C_DIS
LIN {X -0.183,Y -450.221,Z 1347.574,A 0.000,B 0.000,C 90.000,E1 283.355} C_DIS
LIN {X 0.123,Y -453.954,Z 1347.570,A 0.000,B 0.000,C 90.000,E1 282.535} C_DIS
LIN {X 0.018,Y -456.985,Z 1347.565,A 0.000,B 0.000,C 90.000,E1 281.771} C_DIS
LIN {X 0.106,Y -458.568,Z 1347.563,A 0.000,B 0.000,C 90.000,E1 281.243} C_DIS
LIN {X 0.120,Y -459.763,Z 1347.560,A 0.000,B 0.000,C 90.000,E1 280.725} C_DIS
LIN {X -0.223,Y -460.547,Z 1347.557,A 0.000,B 0.000,C 90.000,E1 280.254} C_DIS
LIN {X -0.110,Y -460.854,Z 1347.554,A 0.000,B 0.000,C 90.000,E1 279.726} C_DIS
LIN {X -0.071,Y -460.749,Z 1347.551,A 0.000,B 0.000,C 90.000,E1 279.208} C_DIS
LIN {X 0.044,Y -460.139,Z 1347.548,A 0.000,B 0.000,C 90.000,E1 278.681} C_DIS
LIN {X 0.087,Y -458.996,Z 1347.545,A 0.000,B 0.000,C 90.000,E1 278.163} C_DIS
LIN {X 0.129,Y -457.370,Z 1347.543,A 0.000,B 0.000,C 90.000,E1 277.644} C_DIS
LIN {X 0.166,Y -455.239,Z 1347.540,A 0.000,B 0.000,C 90.000,E1 277.125} C_DIS
LIN {X 0.194,Y -452.561,Z 1347.537,A 0.000,B 0.000,C 90.000,E1 276.606} C_DIS
LIN {X -0.001,Y -451.060,Z 1347.535,A 0.000,B 0.000,C 90.000,E1 276.372} C_DIS
LIN {X -0.003,Y -447.407,Z 1347.532,A 0.000,B 0.000,C 90.000,E1 275.853} C_DIS
LIN {X -0.023,Y -443.103,Z 1347.530,A 0.000,B 0.000,C 90.000,E1 275.334} C_DIS
LIN {X -0.054,Y -437.736,Z 1347.527,A 0.000,B 0.000,C 90.000,E1 274.821} C_DIS
LIN {X -0.209,Y -431.723,Z 1347.524,A 0.000,B 0.000,C 90.000,E1 274.359} C_DIS
LIN {X 0.069,Y -425.494,Z 1347.522,A 0.000,B 0.000,C 90.000,E1 273.898} C_DIS
LIN {X -0.170,Y -419.011,Z 1347.520,A 0.000,B 0.000,C 90.000,E1 273.555} C_DIS
LIN {X -0.096,Y -412.444,Z 1347.518,A 0.000,B 0.000,C 90.000,E1 273.212} C_DIS
LIN {X -0.153,Y -405.771,Z 1347.516,A 0.000,B 0.000,C 90.000,E1 272.922} C_DIS
LIN {X 0.010,Y -398.822,Z 1347.515,A 0.000,B 0.000,C 90.000,E1 272.636} C_DIS
LIN {X 0.025,Y -391.826,Z 1347.513,A 0.000,B 0.000,C 90.000,E1 272.407} C_DIS
LIN {X -0.089,Y -384.589,Z 1347.512,A 0.000,B 0.000,C 90.000,E1 272.236} C_DIS
LIN {X 0.021,Y -377.455,Z 1347.511,A 0.000,B 0.000,C 90.000,E1 272.064} C_DIS
LIN {X -0.078,Y -369.592,Z 1347.511,A 0.000,B 0.000,C 90.000,E1 271.949} C_DIS
LIN {X -0.006,Y -360.112,Z 1347.510,A 0.000,B 0.000,C 90.000,E1 271.835} C_DIS
LIN {X 0.141,Y -345.557,Z 1347.510,A 0.000,B 0.000,C 90.000,E1 271.718} C_DIS
LIN {X 0.082,Y -338.569,Z 1347.510,A 0.000,B 0.000,C 90.000,E1 271.718} C_DIS
LIN {X 0.014,Y -181.309,Z 1347.510,A 0.000,B 0.000,C 90.000,E1 271.718} C_DIS
LIN {X 0.087,Y -181.580,Z 1347.501,A 0.000,B 0.000,C 90.000,E1 270.172} C_DIS
LIN {X 0.045,Y -180.907,Z 1347.475,A 0.000,B 0.000,C 90.000,E1 265.469} C_DIS
LIN {X -0.078,Y -180.743,Z 1347.470,A 0.000,B 0.000,C 90.000,E1 264.666} C_DIS
LIN {X 0.023,Y -178.834,Z 1347.442,A 0.000,B 0.000,C 90.000,E1 259.567} C_DIS
LIN {X 0.057,Y -175.878,Z 1347.414,A 0.000,B 0.000,C 90.000,E1 254.464} C_DIS
LIN {X -0.006,Y -174.538,Z 1347.404,A 0.000,B 0.000,C 90.000,E1 252.779} C_DIS
LIN {X 0.087,Y -171.523,Z 1347.380,A 0.000,B 0.000,C 90.000,E1 248.465} C_DIS
LIN {X 0.072,Y -167.749,Z 1347.357,A 0.000,B 0.000,C 90.000,E1 244.152} C_DIS
LIN {X 0.011,Y -166.451,Z 1347.347,A 0.000,B 0.000,C 90.000,E1 242.436} C_DIS
LIN {X 0.001,Y -163.168,Z 1347.328,A 0.000,B 0.000,C 90.000,E1 238.948} C_DIS
LIN {X 0.050,Y -161.126,Z 1347.313,A 0.000,B 0.000,C 90.000,E1 236.294} C_DIS
LIN {X -0.047,Y -157.148,Z 1347.288,A 0.000,B 0.000,C 90.000,E1 231.904} C_DIS
LIN {X -0.024,Y -155.881,Z 1347.278,A 0.000,B 0.000,C 90.000,E1 230.114} C_DIS
LIN {X -0.065,Y -152.132,Z 1347.253,A 0.000,B 0.000,C 90.000,E1 225.648} C_DIS
LIN {X -0.045,Y -150.381,Z 1347.238,A 0.000,B 0.000,C 90.000,E1 222.933} C_DIS
SetRPM(0)
End
